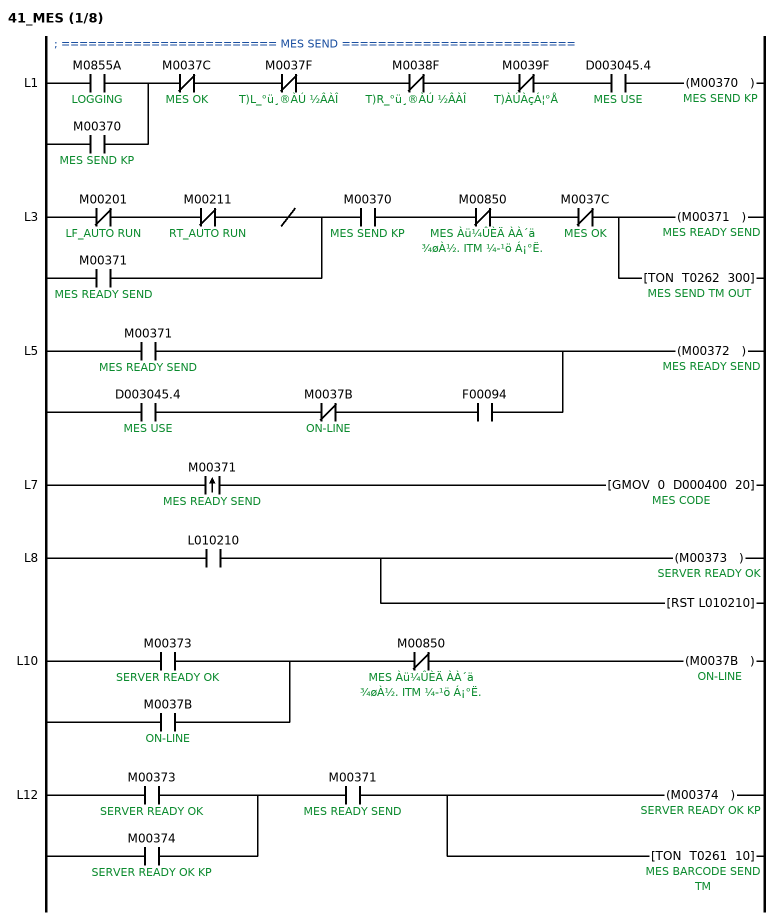
[picture p240: 41_MES rungs L1-L12]
// ======================== MES SEND ==========================
; L1
LOAD      M0855A	// LOGGING
OR        M00370	// MES SEND KP
AND NOT   M0037C	// MES OK
AND NOT   M0037F	// T)L_°ü¸®ÀÚ ½ÂÀÎ
AND NOT   M0038F	// T)R_°ü¸®ÀÚ ½ÂÀÎ
AND NOT   M0039F	// T)ÀÚÀçÁ¦°Å
AND       D003045.4	// MES USE
OUT       M00370	// MES SEND KP
; L3
LOAD NOT  M00201	// LF_AUTO RUN
AND NOT   M00211	// RT_AUTO RUN
NOT
OR        M00371	// MES READY SEND
AND       M00370	// MES SEND KP
AND NOT   M00850	// MES Àü¼ÛÈÄ ÀÀ´ä ¾øÀ½. ITM ¼­¹ö Á¡°Ë.
AND NOT   M0037C	// MES OK
OUT       M00371	// MES READY SEND
TON       T0262 300	// MES SEND TM OUT
; L5
LOAD      M00371	// MES READY SEND
LOAD      D003045.4	// MES USE
AND NOT   M0037B	// ON-LINE
AND       F00094
OR LOAD
OUT       M00372	// MES READY SEND
; L7
LOADP     M00371	// MES READY SEND
GMOV      0 D000400 20	// MES CODE
; L8
LOAD      L010210
OUT       M00373	// SERVER READY OK
RST       L010210
; L10
LOAD      M00373	// SERVER READY OK
OR        M0037B	// ON-LINE
AND NOT   M00850	// MES Àü¼ÛÈÄ ÀÀ´ä ¾øÀ½. ITM ¼­¹ö Á¡°Ë.
OUT       M0037B	// ON-LINE
; L12
LOAD      M00373	// SERVER READY OK
OR        M00374	// SERVER READY OK KP
AND       M00371	// MES READY SEND
OUT       M00374	// SERVER READY OK KP
TON       T0261 10	// MES BARCODE SEND TM

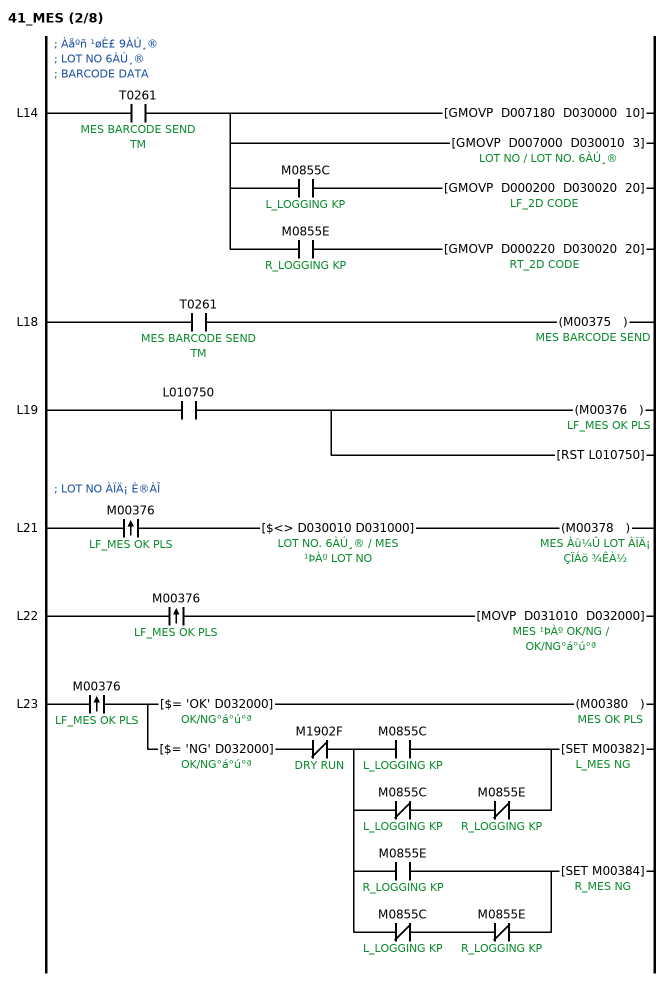
; L14
LOAD      T0261	// MES BARCODE SEND TM
GMOVP     D007180 D030000 10
GMOVP     D007000 D030010 3	// LOT NO / LOT NO. 6ÀÚ¸®
MPUSH
AND       M0855C	// L_LOGGING KP
GMOVP     D000200 D030020 20	// LF_2D CODE
MPOP
AND       M0855E	// R_LOGGING KP
GMOVP     D000220 D030020 20	// RT_2D CODE
// output comment: Àåºñ ¹øÈ£ 9ÀÚ¸®
// output comment: LOT NO 6ÀÚ¸®
// output comment: BARCODE DATA
; L18
LOAD      T0261	// MES BARCODE SEND TM
OUT       M00375	// MES BARCODE SEND
; L19
LOAD      L010750
OUT       M00376	// LF_MES OK PLS
RST       L010750
; L21
LOADP     M00376	// LF_MES OK PLS
AND$<>    D030010 D031000	// LOT NO. 6ÀÚ¸® / MES ¹ÞÀº LOT NO
OUT       M00378	// MES Àü¼Û LOT ÀÏÄ¡ ÇÏÁö ¾ÊÀ½
// output comment: LOT NO ÀÏÄ¡ È®ÀÎ
; L22
LOADP     M00376	// LF_MES OK PLS
MOVP      D031010 D032000	// MES ¹ÞÀº OK/NG / OK/NG°á°ú°ª
; L23
LOADP     M00376	// LF_MES OK PLS
MPUSH
AND$=     'OK' D032000	// OK/NG°á°ú°ª
OUT       M00380	// MES OK PLS
MPOP
AND$=     'NG' D032000	// OK/NG°á°ú°ª
AND NOT   M1902F	// DRY RUN
MPUSH
LOAD      M0855C	// L_LOGGING KP
LOAD NOT  M0855C	// L_LOGGING KP
AND NOT   M0855E	// R_LOGGING KP
OR LOAD
AND LOAD
SET       M00382	// L_MES NG
MPOP
LOAD      M0855E	// R_LOGGING KP
LOAD NOT  M0855C	// L_LOGGING KP
AND NOT   M0855E	// R_LOGGING KP
OR LOAD
AND LOAD
SET       M00384	// R_MES NG

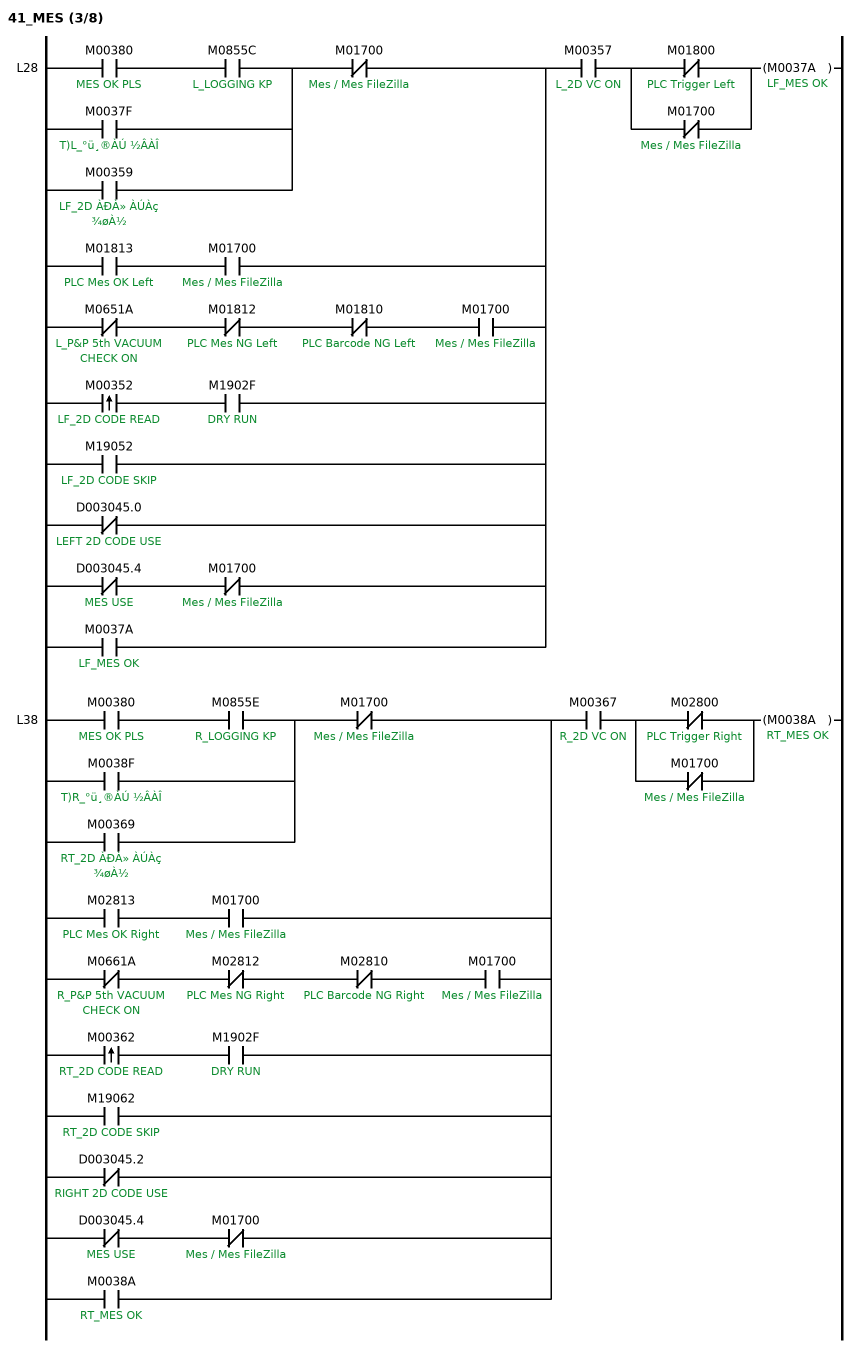
; L28
LOAD      M00380	// MES OK PLS
AND       M0855C	// L_LOGGING KP
OR        M0037F	// T)L_°ü¸®ÀÚ ½ÂÀÎ
OR        M00359	// LF_2D ÀÐÀ» ÀÚÀç ¾øÀ½
AND NOT   M01700	// Mes / Mes FileZilla
LOAD      M01813	// PLC Mes OK Left
AND       M01700	// Mes / Mes FileZilla
OR LOAD
LOAD NOT  M0651A	// L_P&P 5th VACUUM CHECK ON
AND NOT   M01812	// PLC Mes NG Left
AND NOT   M01810	// PLC Barcode NG Left
AND       M01700	// Mes / Mes FileZilla
OR LOAD
LOADP     M00352	// LF_2D CODE READ
AND       M1902F	// DRY RUN
OR LOAD
OR        M19052	// LF_2D CODE SKIP
OR NOT    D003045.0	// LEFT 2D CODE USE
LOAD NOT  D003045.4	// MES USE
AND NOT   M01700	// Mes / Mes FileZilla
OR LOAD
OR        M0037A	// LF_MES OK
AND       M00357	// L_2D VC ON
LOAD NOT  M01800	// PLC Trigger Left
OR NOT    M01700	// Mes / Mes FileZilla
AND LOAD
OUT       M0037A	// LF_MES OK
; L38
LOAD      M00380	// MES OK PLS
AND       M0855E	// R_LOGGING KP
OR        M0038F	// T)R_°ü¸®ÀÚ ½ÂÀÎ
OR        M00369	// RT_2D ÀÐÀ» ÀÚÀç ¾øÀ½
AND NOT   M01700	// Mes / Mes FileZilla
LOAD      M02813	// PLC Mes OK Right
AND       M01700	// Mes / Mes FileZilla
OR LOAD
LOAD NOT  M0661A	// R_P&P 5th VACUUM CHECK ON
AND NOT   M02812	// PLC Mes NG Right
AND NOT   M02810	// PLC Barcode NG Right
AND       M01700	// Mes / Mes FileZilla
OR LOAD
LOADP     M00362	// RT_2D CODE READ
AND       M1902F	// DRY RUN
OR LOAD
OR        M19062	// RT_2D CODE SKIP
OR NOT    D003045.2	// RIGHT 2D CODE USE
LOAD NOT  D003045.4	// MES USE
AND NOT   M01700	// Mes / Mes FileZilla
OR LOAD
OR        M0038A	// RT_MES OK
AND       M00367	// R_2D VC ON
LOAD NOT  M02800	// PLC Trigger Right
OR NOT    M01700	// Mes / Mes FileZilla
AND LOAD
OUT       M0038A	// RT_MES OK

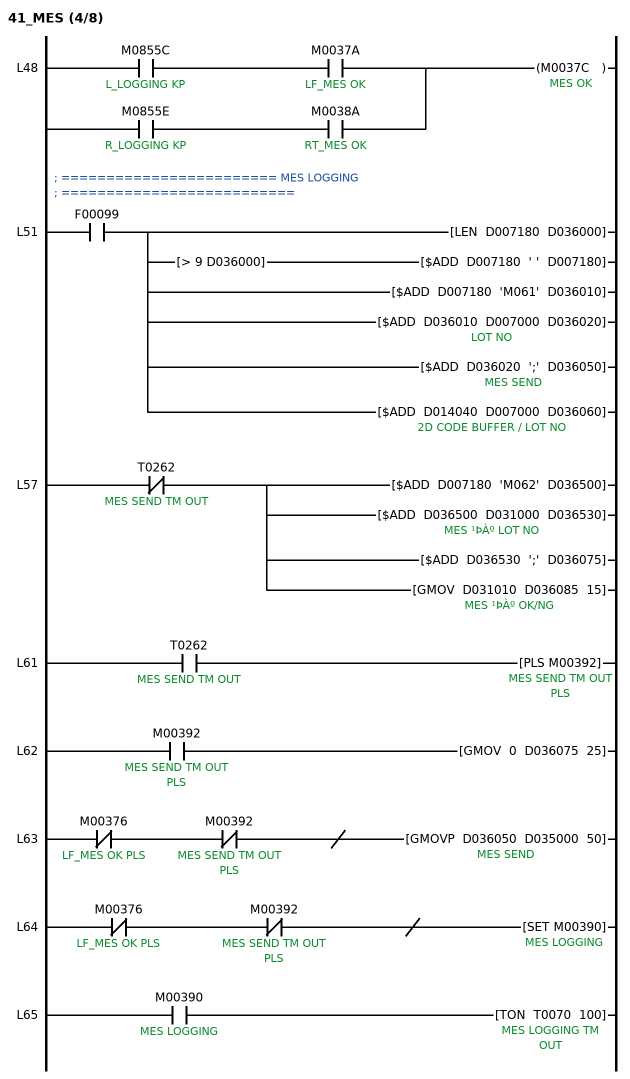
; L48
LOAD      M0855C	// L_LOGGING KP
AND       M0037A	// LF_MES OK
LOAD      M0855E	// R_LOGGING KP
AND       M0038A	// RT_MES OK
OR LOAD
OUT       M0037C	// MES OK
// ======================== MES LOGGING ==========================
; L51
LOAD      F00099
LEN       D007180 D036000
MPUSH
AND>      9 D036000
$ADD      D007180 ' ' D007180
MPOP
$ADD      D007180 'M061' D036010
$ADD      D036010 D007000 D036020	// LOT NO
$ADD      D036020 ';' D036050	// MES SEND
$ADD      D014040 D007000 D036060	// 2D CODE BUFFER / LOT NO
; L57
LOAD NOT  T0262	// MES SEND TM OUT
$ADD      D007180 'M062' D036500
$ADD      D036500 D031000 D036530	// MES ¹ÞÀº LOT NO
$ADD      D036530 ';' D036075
GMOV      D031010 D036085 15	// MES ¹ÞÀº OK/NG
; L61
LOAD      T0262	// MES SEND TM OUT
OUTP      M00392	// MES SEND TM OUT PLS
; L62
LOAD      M00392	// MES SEND TM OUT PLS
GMOV      0 D036075 25
; L63
LOAD NOT  M00376	// LF_MES OK PLS
AND NOT   M00392	// MES SEND TM OUT PLS
NOT
GMOVP     D036050 D035000 50	// MES SEND
; L64
LOAD NOT  M00376	// LF_MES OK PLS
AND NOT   M00392	// MES SEND TM OUT PLS
NOT
SET       M00390	// MES LOGGING
; L65
LOAD      M00390	// MES LOGGING
TON       T0070 100	// MES LOGGING TM OUT

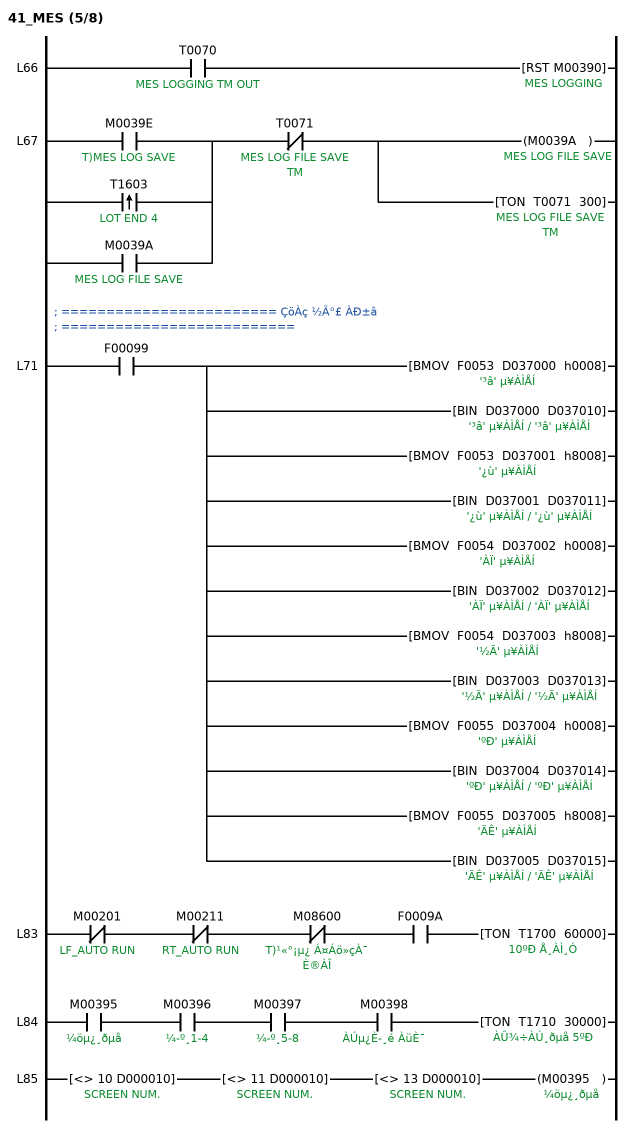
; L66
LOAD      T0070	// MES LOGGING TM OUT
RST       M00390	// MES LOGGING
; L67
LOAD      M0039E	// T)MES LOG SAVE
ORP       T1603	// LOT END 4
OR        M0039A	// MES LOG FILE SAVE
AND NOT   T0071	// MES LOG FILE SAVE TM
OUT       M0039A	// MES LOG FILE SAVE
TON       T0071 300	// MES LOG FILE SAVE TM
// ======================== ÇöÀç ½Ã°£ ÀÐ±â ==========================
; L71
LOAD      F00099
BMOV      F0053 D037000 h0008	// '³â' µ¥ÀÌÅÍ
BIN       D037000 D037010	// '³â' µ¥ÀÌÅÍ / '³â' µ¥ÀÌÅÍ
BMOV      F0053 D037001 h8008	// '¿ù' µ¥ÀÌÅÍ
BIN       D037001 D037011	// '¿ù' µ¥ÀÌÅÍ / '¿ù' µ¥ÀÌÅÍ
BMOV      F0054 D037002 h0008	// 'ÀÏ' µ¥ÀÌÅÍ
BIN       D037002 D037012	// 'ÀÏ' µ¥ÀÌÅÍ / 'ÀÏ' µ¥ÀÌÅÍ
BMOV      F0054 D037003 h8008	// '½Ã' µ¥ÀÌÅÍ
BIN       D037003 D037013	// '½Ã' µ¥ÀÌÅÍ / '½Ã' µ¥ÀÌÅÍ
BMOV      F0055 D037004 h0008	// 'ºÐ' µ¥ÀÌÅÍ
BIN       D037004 D037014	// 'ºÐ' µ¥ÀÌÅÍ / 'ºÐ' µ¥ÀÌÅÍ
BMOV      F0055 D037005 h8008	// 'ÃÊ' µ¥ÀÌÅÍ
BIN       D037005 D037015	// 'ÃÊ' µ¥ÀÌÅÍ / 'ÃÊ' µ¥ÀÌÅÍ
; L83
LOAD NOT  M00201	// LF_AUTO RUN
AND NOT   M00211	// RT_AUTO RUN
AND NOT   M08600	// T)¹«°¡µ¿ Á¤Áö»çÀ¯ È®ÀÎ
AND       F0009A
TON       T1700 60000	// 10ºÐ Å¸ÀÌ¸Ó
; L84
LOAD      M00395	// ¼öµ¿¸ðµå
AND       M00396	// ¼­º¸1-4
AND       M00397	// ¼­º¸5-8
AND       M00398	// ÀÚµ¿È­¸é ÀüÈ¯
TON       T1710 30000	// ÀÛ¾÷ÀÚ¸ðµå 5ºÐ
; L85
LOAD<>    10 D000010	// SCREEN NUM.
AND<>     11 D000010	// SCREEN NUM.
AND<>     13 D000010	// SCREEN NUM.
OUT       M00395	// ¼öµ¿¸ðµå

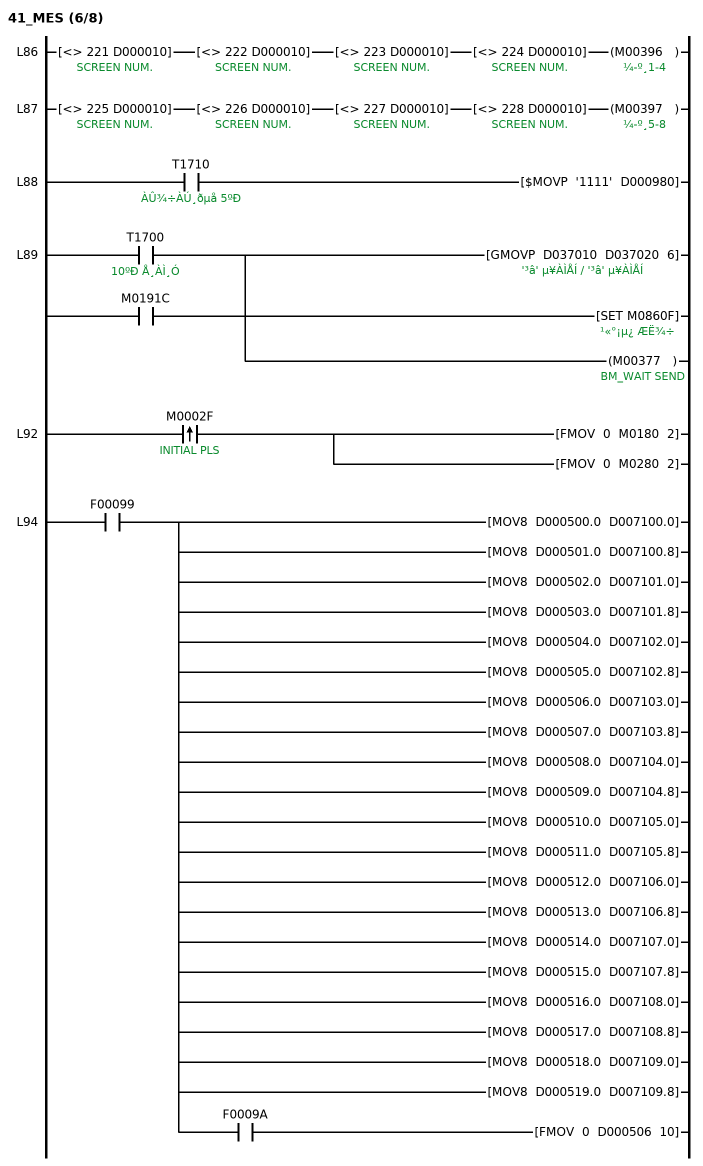
; L86
LOAD<>    221 D000010	// SCREEN NUM.
AND<>     222 D000010	// SCREEN NUM.
AND<>     223 D000010	// SCREEN NUM.
AND<>     224 D000010	// SCREEN NUM.
OUT       M00396	// ¼­º¸1-4
; L87
LOAD<>    225 D000010	// SCREEN NUM.
AND<>     226 D000010	// SCREEN NUM.
AND<>     227 D000010	// SCREEN NUM.
AND<>     228 D000010	// SCREEN NUM.
OUT       M00397	// ¼­º¸5-8
; L88
LOAD      T1710	// ÀÛ¾÷ÀÚ¸ðµå 5ºÐ
$MOVP     '1111' D000980
; L89
LOAD      T1700	// 10ºÐ Å¸ÀÌ¸Ó
OR        M0191C
GMOVP     D037010 D037020 6	// '³â' µ¥ÀÌÅÍ / '³â' µ¥ÀÌÅÍ
SET       M0860F	// ¹«°¡µ¿ ÆË¾÷
OUT       M00377	// BM_WAIT SEND
; L92
LOADP     M0002F	// INITIAL PLS
FMOV      0 M0180 2
FMOV      0 M0280 2
; L94
LOAD      F00099
MOV8      D000500.0 D007100.0
MOV8      D000501.0 D007100.8
MOV8      D000502.0 D007101.0
MOV8      D000503.0 D007101.8
MOV8      D000504.0 D007102.0
MOV8      D000505.0 D007102.8
MOV8      D000506.0 D007103.0
MOV8      D000507.0 D007103.8
MOV8      D000508.0 D007104.0
MOV8      D000509.0 D007104.8
MOV8      D000510.0 D007105.0
MOV8      D000511.0 D007105.8
MOV8      D000512.0 D007106.0
MOV8      D000513.0 D007106.8
MOV8      D000514.0 D007107.0
MOV8      D000515.0 D007107.8
MOV8      D000516.0 D007108.0
MOV8      D000517.0 D007108.8
MOV8      D000518.0 D007109.0
MOV8      D000519.0 D007109.8
AND       F0009A
FMOV      0 D000506 10

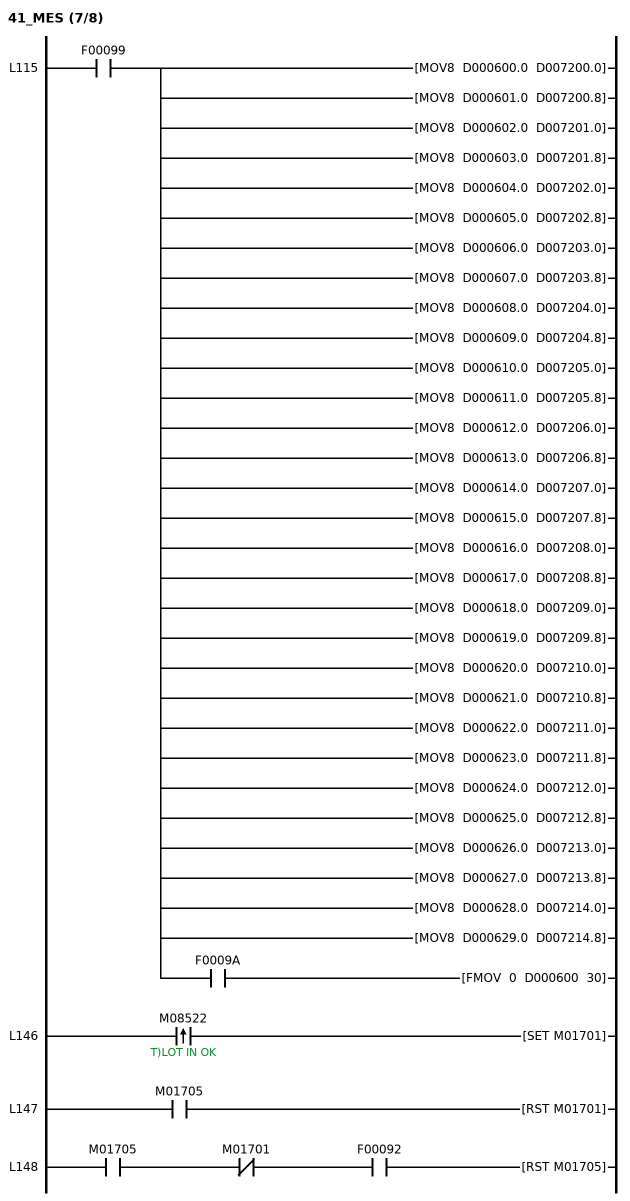
; L115
LOAD      F00099
MOV8      D000600.0 D007200.0
MOV8      D000601.0 D007200.8
MOV8      D000602.0 D007201.0
MOV8      D000603.0 D007201.8
MOV8      D000604.0 D007202.0
MOV8      D000605.0 D007202.8
MOV8      D000606.0 D007203.0
MOV8      D000607.0 D007203.8
MOV8      D000608.0 D007204.0
MOV8      D000609.0 D007204.8
MOV8      D000610.0 D007205.0
MOV8      D000611.0 D007205.8
MOV8      D000612.0 D007206.0
MOV8      D000613.0 D007206.8
MOV8      D000614.0 D007207.0
MOV8      D000615.0 D007207.8
MOV8      D000616.0 D007208.0
MOV8      D000617.0 D007208.8
MOV8      D000618.0 D007209.0
MOV8      D000619.0 D007209.8
MOV8      D000620.0 D007210.0
MOV8      D000621.0 D007210.8
MOV8      D000622.0 D007211.0
MOV8      D000623.0 D007211.8
MOV8      D000624.0 D007212.0
MOV8      D000625.0 D007212.8
MOV8      D000626.0 D007213.0
MOV8      D000627.0 D007213.8
MOV8      D000628.0 D007214.0
MOV8      D000629.0 D007214.8
AND       F0009A
FMOV      0 D000600 30
; L146
LOADP     M08522	// T)LOT IN OK
SET       M01701
; L147
LOAD      M01705
RST       M01701
; L148
LOAD      M01705
AND NOT   M01701
AND       F00092
RST       M01705

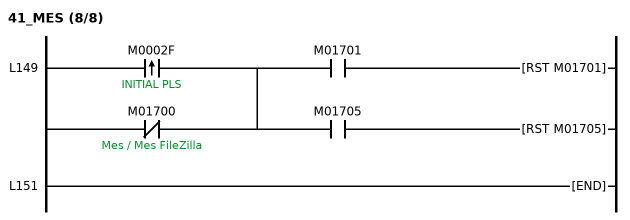
; L149
LOADP     M0002F	// INITIAL PLS
OR NOT    M01700	// Mes / Mes FileZilla
MPUSH
AND       M01701
RST       M01701
MPOP
AND       M01705
RST       M01705
; L151
END

PROGRAM 51_MT_01_2_3_4 (task: ½ºÄµ ÇÁ·Î±×·¥)

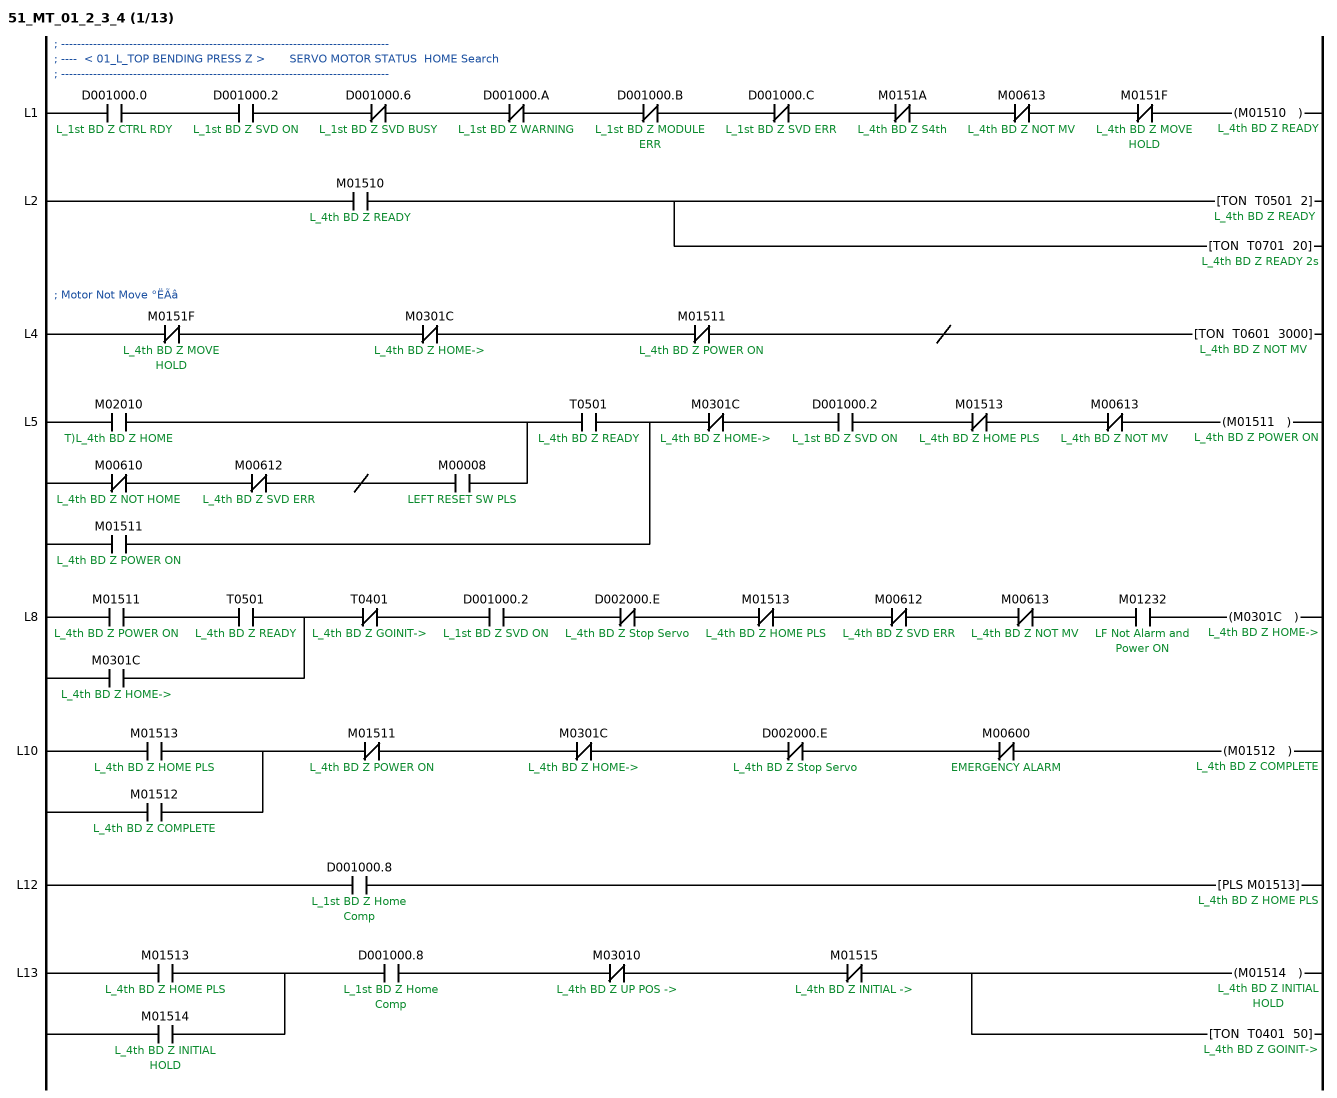
// ----------------------------------------------------------------------------------
// 
// ----  < 01_L_TOP BENDING PRESS Z >       SERVO MOTOR STATUS  HOME Search
// 
// ----------------------------------------------------------------------------------
; L1
LOAD      D001000.0	// L_1st BD Z CTRL RDY
AND       D001000.2	// L_1st BD Z SVD ON
AND NOT   D001000.6	// L_1st BD Z SVD BUSY
AND NOT   D001000.A	// L_1st BD Z WARNING
AND NOT   D001000.B	// L_1st BD Z MODULE ERR
AND NOT   D001000.C	// L_1st BD Z SVD ERR
AND NOT   M0151A	// L_4th BD Z S4th
AND NOT   M00613	// L_4th BD Z NOT MV
AND NOT   M0151F	// L_4th BD Z MOVE HOLD
OUT       M01510	// L_4th BD Z READY
; L2
LOAD      M01510	// L_4th BD Z READY
TON       T0501 2	// L_4th BD Z READY
TON       T0701 20	// L_4th BD Z READY 2s
; L4
LOAD NOT  M0151F	// L_4th BD Z MOVE HOLD
AND NOT   M0301C	// L_4th BD Z HOME->
AND NOT   M01511	// L_4th BD Z POWER ON
NOT
TON       T0601 3000	// L_4th BD Z NOT MV
// output comment: Motor Not Move °ËÃâ
; L5
LOAD      M02010	// T)L_4th BD Z HOME
LOAD NOT  M00610	// L_4th BD Z NOT HOME
AND NOT   M00612	// L_4th BD Z SVD ERR
NOT
AND       M00008	// LEFT RESET SW PLS
OR LOAD
AND       T0501	// L_4th BD Z READY
OR        M01511	// L_4th BD Z POWER ON
AND NOT   M0301C	// L_4th BD Z HOME->
AND       D001000.2	// L_1st BD Z SVD ON
AND NOT   M01513	// L_4th BD Z HOME PLS
AND NOT   M00613	// L_4th BD Z NOT MV
OUT       M01511	// L_4th BD Z POWER ON
; L8
LOAD      M01511	// L_4th BD Z POWER ON
AND       T0501	// L_4th BD Z READY
OR        M0301C	// L_4th BD Z HOME->
AND NOT   T0401	// L_4th BD Z GOINIT->
AND       D001000.2	// L_1st BD Z SVD ON
AND NOT   D002000.E	// L_4th BD Z Stop Servo
AND NOT   M01513	// L_4th BD Z HOME PLS
AND NOT   M00612	// L_4th BD Z SVD ERR
AND NOT   M00613	// L_4th BD Z NOT MV
AND       M01232	// LF Not Alarm and Power ON
OUT       M0301C	// L_4th BD Z HOME->
; L10
LOAD      M01513	// L_4th BD Z HOME PLS
OR        M01512	// L_4th BD Z COMPLETE
AND NOT   M01511	// L_4th BD Z POWER ON
AND NOT   M0301C	// L_4th BD Z HOME->
AND NOT   D002000.E	// L_4th BD Z Stop Servo
AND NOT   M00600	// EMERGENCY ALARM
OUT       M01512	// L_4th BD Z COMPLETE
; L12
LOAD      D001000.8	// L_1st BD Z Home Comp
OUTP      M01513	// L_4th BD Z HOME PLS
; L13
LOAD      M01513	// L_4th BD Z HOME PLS
OR        M01514	// L_4th BD Z INITIAL HOLD
AND       D001000.8	// L_1st BD Z Home Comp
AND NOT   M03010	// L_4th BD Z UP POS ->
AND NOT   M01515	// L_4th BD Z INITIAL ->
OUT       M01514	// L_4th BD Z INITIAL HOLD
TON       T0401 50	// L_4th BD Z GOINIT->

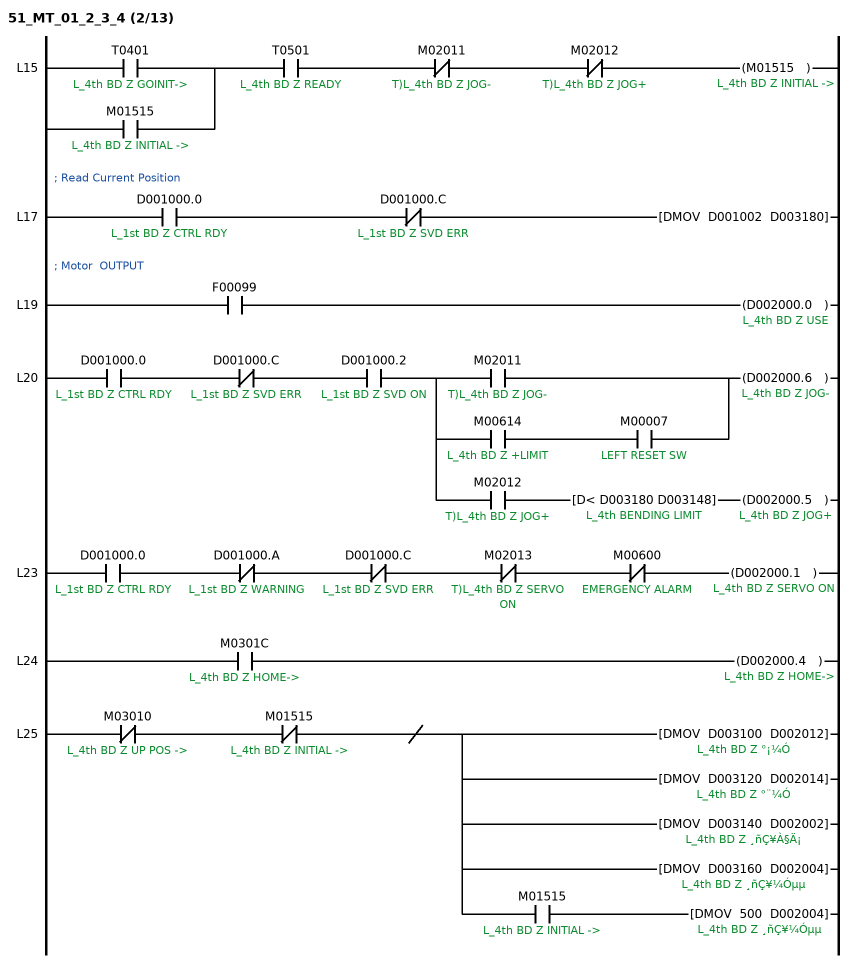
; L15
LOAD      T0401	// L_4th BD Z GOINIT->
OR        M01515	// L_4th BD Z INITIAL ->
AND       T0501	// L_4th BD Z READY
AND NOT   M02011	// T)L_4th BD Z JOG-
AND NOT   M02012	// T)L_4th BD Z JOG+
OUT       M01515	// L_4th BD Z INITIAL ->
; L17
LOAD      D001000.0	// L_1st BD Z CTRL RDY
AND NOT   D001000.C	// L_1st BD Z SVD ERR
DMOV      D001002 D003180
// output comment: Read Current Position
//  Motor  OUTPUT
; L19
LOAD      F00099
OUT       D002000.0	// L_4th BD Z USE
; L20
LOAD      D001000.0	// L_1st BD Z CTRL RDY
AND NOT   D001000.C	// L_1st BD Z SVD ERR
AND       D001000.2	// L_1st BD Z SVD ON
MPUSH
LOAD      M02011	// T)L_4th BD Z JOG-
LOAD      M00614	// L_4th BD Z +LIMIT
AND       M00007	// LEFT RESET SW
OR LOAD
AND LOAD
OUT       D002000.6	// L_4th BD Z JOG-
MPOP
AND       M02012	// T)L_4th BD Z JOG+
ANDD<     D003180 D003148	// L_4th BENDING LIMIT
OUT       D002000.5	// L_4th BD Z JOG+
; L23
LOAD      D001000.0	// L_1st BD Z CTRL RDY
AND NOT   D001000.A	// L_1st BD Z WARNING
AND NOT   D001000.C	// L_1st BD Z SVD ERR
AND NOT   M02013	// T)L_4th BD Z SERVO ON
AND NOT   M00600	// EMERGENCY ALARM
OUT       D002000.1	// L_4th BD Z SERVO ON
; L24
LOAD      M0301C	// L_4th BD Z HOME->
OUT       D002000.4	// L_4th BD Z HOME->
; L25
LOAD NOT  M03010	// L_4th BD Z UP POS ->
AND NOT   M01515	// L_4th BD Z INITIAL ->
NOT
DMOV      D003100 D002012	// L_4th BD Z °¡¼Ó
DMOV      D003120 D002014	// L_4th BD Z °¨¼Ó
DMOV      D003140 D002002	// L_4th BD Z ¸ñÇ¥À§Ä¡
DMOV      D003160 D002004	// L_4th BD Z ¸ñÇ¥¼Óµµ
AND       M01515	// L_4th BD Z INITIAL ->
DMOV      500 D002004	// L_4th BD Z ¸ñÇ¥¼Óµµ

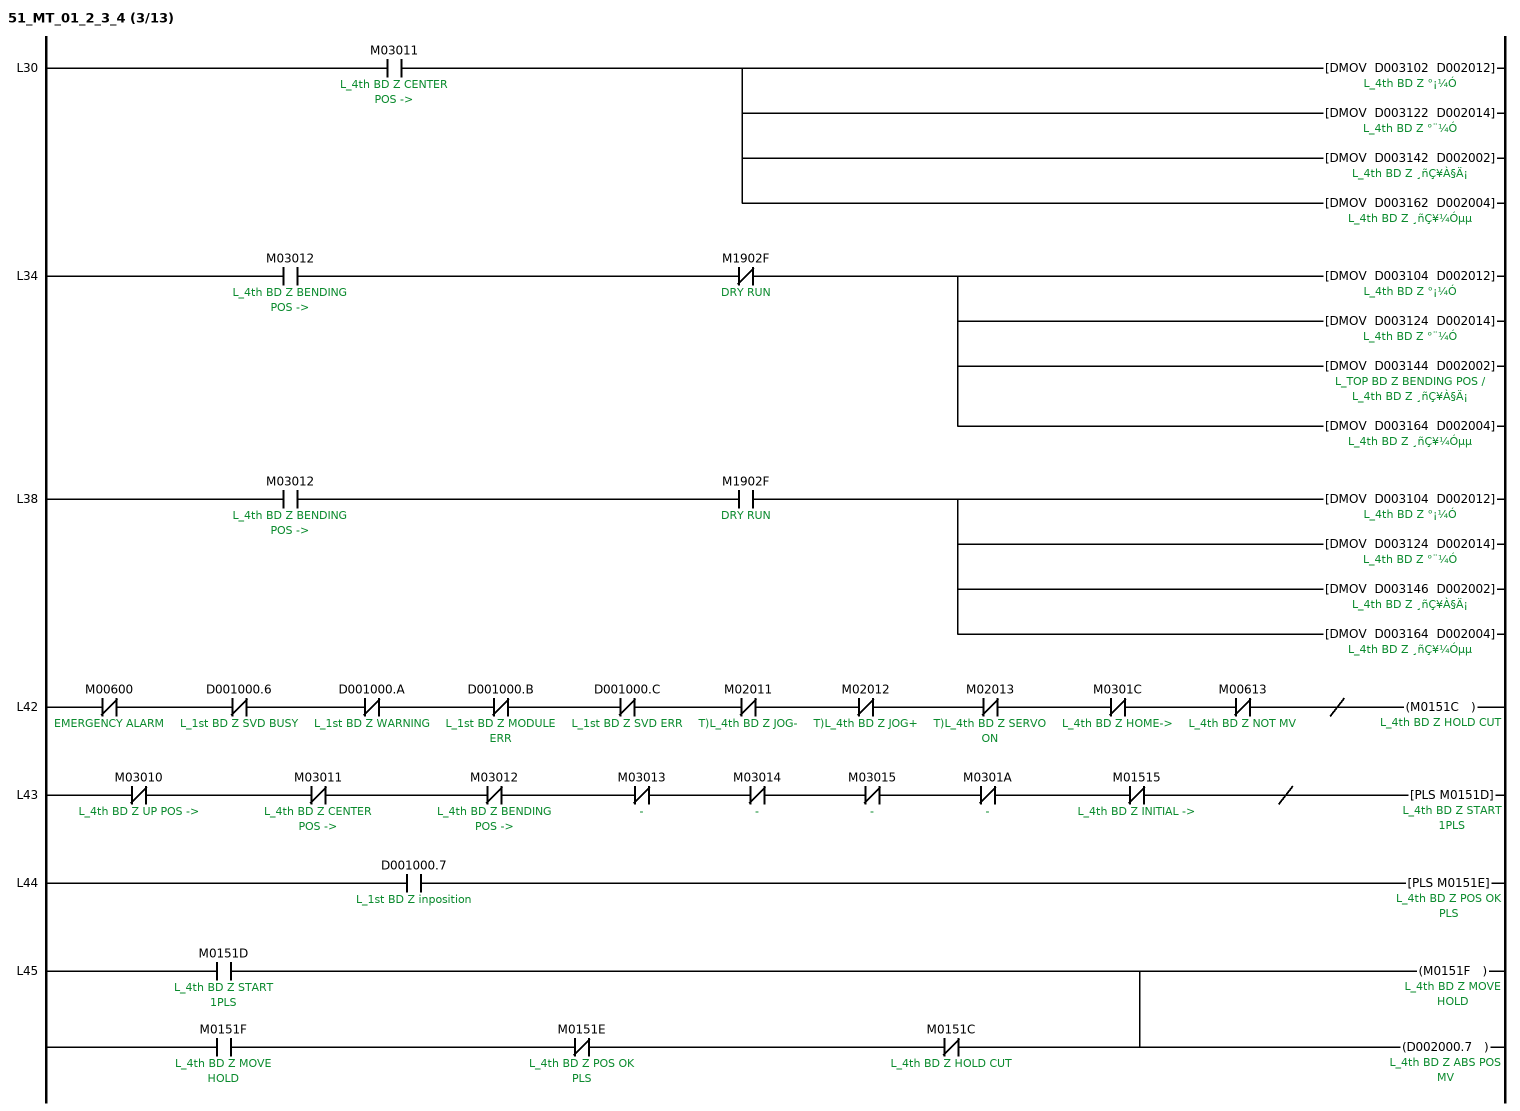
; L30
LOAD      M03011	// L_4th BD Z CENTER POS ->
DMOV      D003102 D002012	// L_4th BD Z °¡¼Ó
DMOV      D003122 D002014	// L_4th BD Z °¨¼Ó
DMOV      D003142 D002002	// L_4th BD Z ¸ñÇ¥À§Ä¡
DMOV      D003162 D002004	// L_4th BD Z ¸ñÇ¥¼Óµµ
; L34
LOAD      M03012	// L_4th BD Z BENDING POS ->
AND NOT   M1902F	// DRY RUN
DMOV      D003104 D002012	// L_4th BD Z °¡¼Ó
DMOV      D003124 D002014	// L_4th BD Z °¨¼Ó
DMOV      D003144 D002002	// L_TOP BD Z BENDING POS / L_4th BD Z ¸ñÇ¥À§Ä¡
DMOV      D003164 D002004	// L_4th BD Z ¸ñÇ¥¼Óµµ
; L38
LOAD      M03012	// L_4th BD Z BENDING POS ->
AND       M1902F	// DRY RUN
DMOV      D003104 D002012	// L_4th BD Z °¡¼Ó
DMOV      D003124 D002014	// L_4th BD Z °¨¼Ó
DMOV      D003146 D002002	// L_4th BD Z ¸ñÇ¥À§Ä¡
DMOV      D003164 D002004	// L_4th BD Z ¸ñÇ¥¼Óµµ
; L42
LOAD NOT  M00600	// EMERGENCY ALARM
AND NOT   D001000.6	// L_1st BD Z SVD BUSY
AND NOT   D001000.A	// L_1st BD Z WARNING
AND NOT   D001000.B	// L_1st BD Z MODULE ERR
AND NOT   D001000.C	// L_1st BD Z SVD ERR
AND NOT   M02011	// T)L_4th BD Z JOG-
AND NOT   M02012	// T)L_4th BD Z JOG+
AND NOT   M02013	// T)L_4th BD Z SERVO ON
AND NOT   M0301C	// L_4th BD Z HOME->
AND NOT   M00613	// L_4th BD Z NOT MV
NOT
OUT       M0151C	// L_4th BD Z HOLD CUT
; L43
LOAD NOT  M03010	// L_4th BD Z UP POS ->
AND NOT   M03011	// L_4th BD Z CENTER POS ->
AND NOT   M03012	// L_4th BD Z BENDING POS ->
AND NOT   M03013	// -
AND NOT   M03014	// -
AND NOT   M03015	// -
AND NOT   M0301A	// -
AND NOT   M01515	// L_4th BD Z INITIAL ->
NOT
OUTP      M0151D	// L_4th BD Z START 1PLS
; L44
LOAD      D001000.7	// L_1st BD Z inposition
OUTP      M0151E	// L_4th BD Z POS OK PLS
; L45
LOAD      M0151D	// L_4th BD Z START 1PLS
LOAD      M0151F	// L_4th BD Z MOVE HOLD
AND NOT   M0151E	// L_4th BD Z POS OK PLS
AND NOT   M0151C	// L_4th BD Z HOLD CUT
OR LOAD
OUT       M0151F	// L_4th BD Z MOVE HOLD
OUT       D002000.7	// L_4th BD Z ABS POS MV

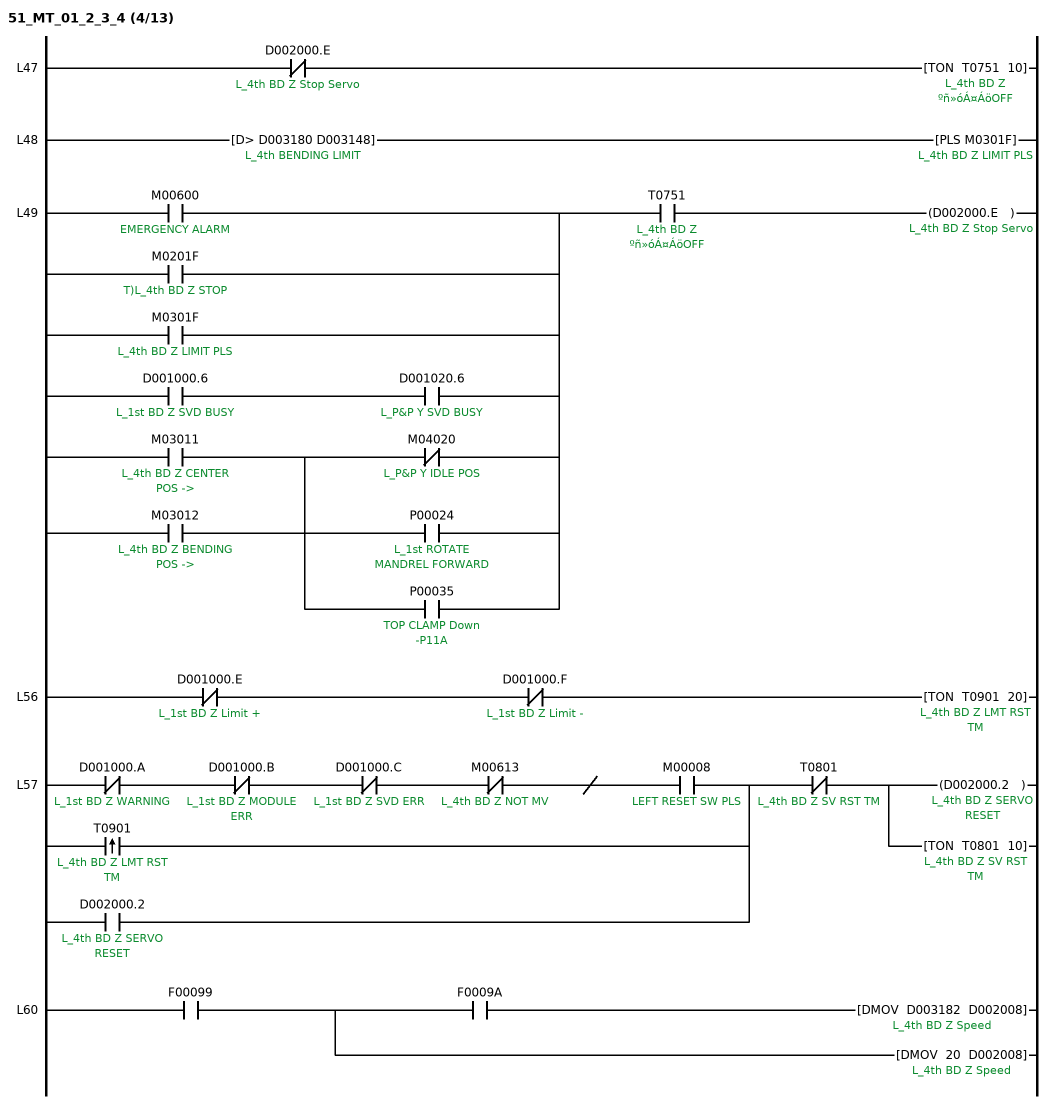
; L47
LOAD NOT  D002000.E	// L_4th BD Z Stop Servo
TON       T0751 10	// L_4th BD Z ºñ»óÁ¤ÁöOFF
; L48
LOADD>    D003180 D003148	// L_4th BENDING LIMIT
OUTP      M0301F	// L_4th BD Z LIMIT PLS
; L49
LOAD      M00600	// EMERGENCY ALARM
OR        M0201F	// T)L_4th BD Z STOP
OR        M0301F	// L_4th BD Z LIMIT PLS
LOAD      D001000.6	// L_1st BD Z SVD BUSY
AND       D001020.6	// L_P&P Y SVD BUSY
OR LOAD
LOAD      M03011	// L_4th BD Z CENTER POS ->
OR        M03012	// L_4th BD Z BENDING POS ->
LOAD NOT  M04020	// L_P&P Y IDLE POS
OR        P00024	// L_1st ROTATE MANDREL FORWARD
OR        P00035	// TOP CLAMP Down -P11A
AND LOAD
OR LOAD
AND       T0751	// L_4th BD Z ºñ»óÁ¤ÁöOFF
OUT       D002000.E	// L_4th BD Z Stop Servo
; L56
LOAD NOT  D001000.E	// L_1st BD Z Limit +
AND NOT   D001000.F	// L_1st BD Z Limit -
TON       T0901 20	// L_4th BD Z LMT RST TM
; L57
LOAD NOT  D001000.A	// L_1st BD Z WARNING
AND NOT   D001000.B	// L_1st BD Z MODULE ERR
AND NOT   D001000.C	// L_1st BD Z SVD ERR
AND NOT   M00613	// L_4th BD Z NOT MV
NOT
AND       M00008	// LEFT RESET SW PLS
ORP       T0901	// L_4th BD Z LMT RST TM
OR        D002000.2	// L_4th BD Z SERVO RESET
AND NOT   T0801	// L_4th BD Z SV RST TM
OUT       D002000.2	// L_4th BD Z SERVO RESET
TON       T0801 10	// L_4th BD Z SV RST TM
; L60
LOAD      F00099
MPUSH
AND       F0009A
DMOV      D003182 D002008	// L_4th BD Z Speed
MPOP
DMOV      20 D002008	// L_4th BD Z Speed

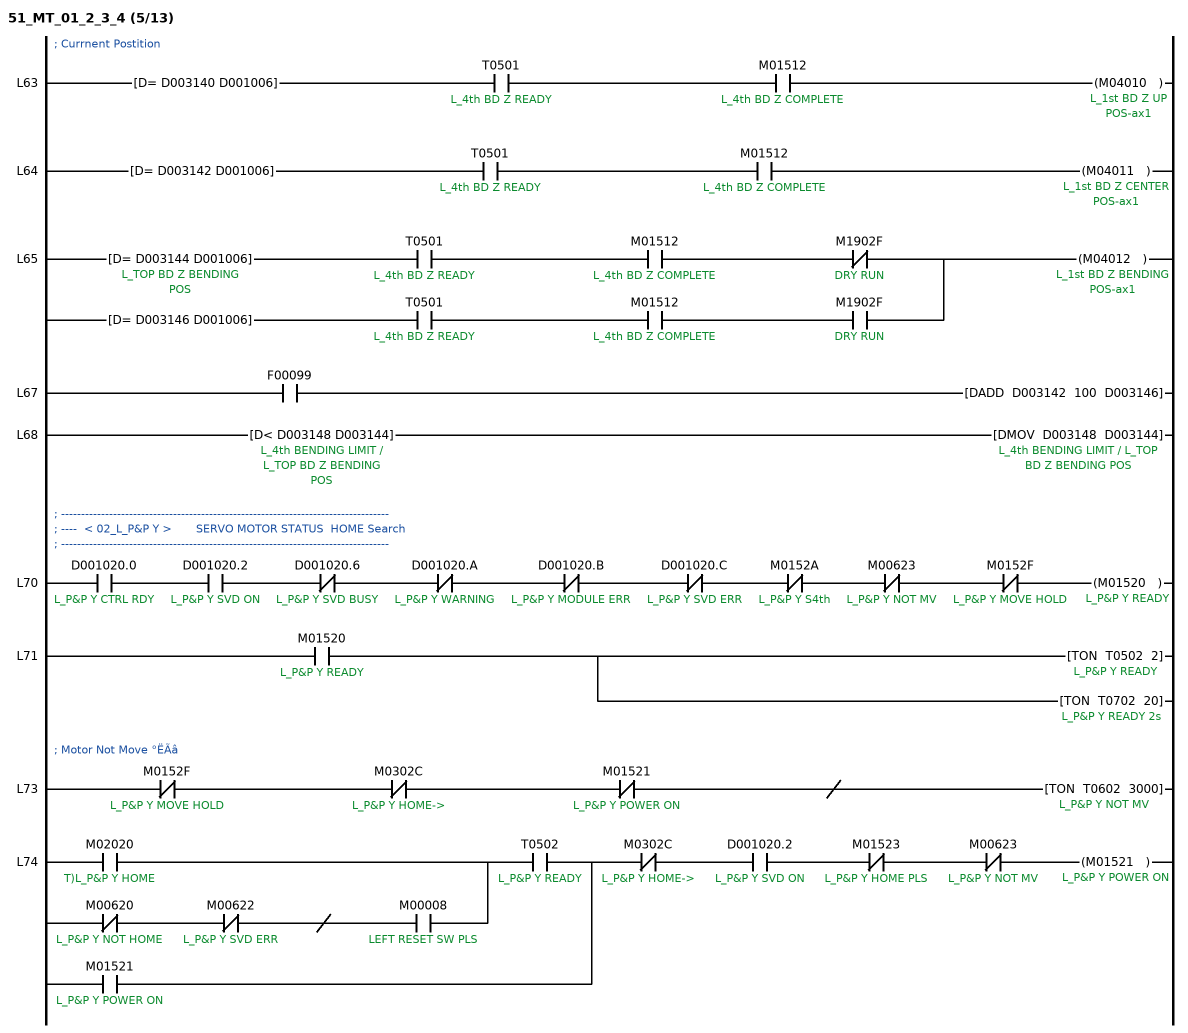
// Currnent Postition
; L63
LOADD=    D003140 D001006
AND       T0501	// L_4th BD Z READY
AND       M01512	// L_4th BD Z COMPLETE
OUT       M04010	// L_1st BD Z UP POS-ax1
; L64
LOADD=    D003142 D001006
AND       T0501	// L_4th BD Z READY
AND       M01512	// L_4th BD Z COMPLETE
OUT       M04011	// L_1st BD Z CENTER POS-ax1
; L65
LOADD=    D003144 D001006	// L_TOP BD Z BENDING POS
AND       T0501	// L_4th BD Z READY
AND       M01512	// L_4th BD Z COMPLETE
AND NOT   M1902F	// DRY RUN
LOADD=    D003146 D001006
AND       T0501	// L_4th BD Z READY
AND       M01512	// L_4th BD Z COMPLETE
AND       M1902F	// DRY RUN
OR LOAD
OUT       M04012	// L_1st BD Z BENDING POS-ax1
; L67
LOAD      F00099
DADD      D003142 100 D003146
; L68
LOADD<    D003148 D003144	// L_4th BENDING LIMIT / L_TOP BD Z BENDING POS
DMOV      D003148 D003144	// L_4th BENDING LIMIT / L_TOP BD Z BENDING POS
// ----------------------------------------------------------------------------------
// 
// ----  < 02_L_P&P Y >       SERVO MOTOR STATUS  HOME Search
// 
// ----------------------------------------------------------------------------------
; L70
LOAD      D001020.0	// L_P&P Y CTRL RDY
AND       D001020.2	// L_P&P Y SVD ON
AND NOT   D001020.6	// L_P&P Y SVD BUSY
AND NOT   D001020.A	// L_P&P Y WARNING
AND NOT   D001020.B	// L_P&P Y MODULE ERR
AND NOT   D001020.C	// L_P&P Y SVD ERR
AND NOT   M0152A	// L_P&P Y S4th
AND NOT   M00623	// L_P&P Y NOT MV
AND NOT   M0152F	// L_P&P Y MOVE HOLD
OUT       M01520	// L_P&P Y READY
; L71
LOAD      M01520	// L_P&P Y READY
TON       T0502 2	// L_P&P Y READY
TON       T0702 20	// L_P&P Y READY 2s
; L73
LOAD NOT  M0152F	// L_P&P Y MOVE HOLD
AND NOT   M0302C	// L_P&P Y HOME->
AND NOT   M01521	// L_P&P Y POWER ON
NOT
TON       T0602 3000	// L_P&P Y NOT MV
// output comment: Motor Not Move °ËÃâ
; L74
LOAD      M02020	// T)L_P&P Y HOME
LOAD NOT  M00620	// L_P&P Y NOT HOME
AND NOT   M00622	// L_P&P Y SVD ERR
NOT
AND       M00008	// LEFT RESET SW PLS
OR LOAD
AND       T0502	// L_P&P Y READY
OR        M01521	// L_P&P Y POWER ON
AND NOT   M0302C	// L_P&P Y HOME->
AND       D001020.2	// L_P&P Y SVD ON
AND NOT   M01523	// L_P&P Y HOME PLS
AND NOT   M00623	// L_P&P Y NOT MV
OUT       M01521	// L_P&P Y POWER ON

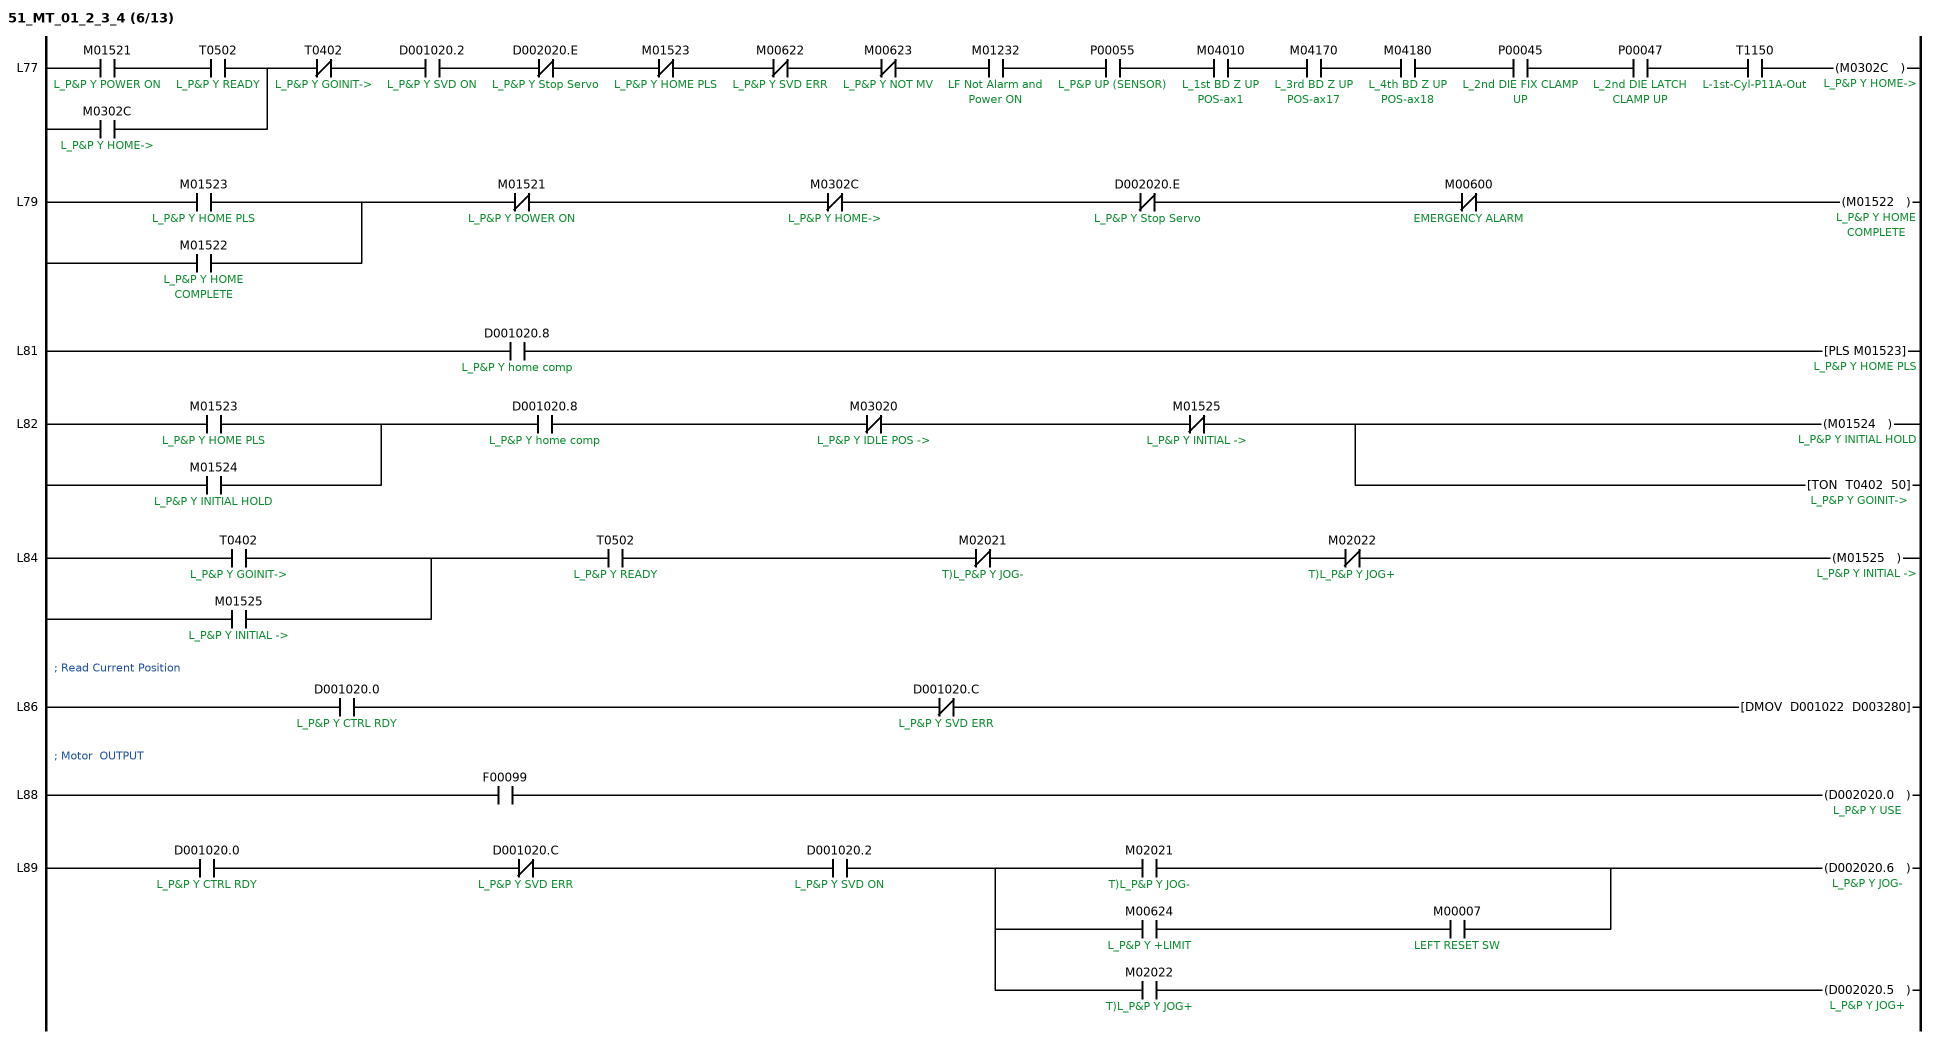
; L77
LOAD      M01521	// L_P&P Y POWER ON
AND       T0502	// L_P&P Y READY
OR        M0302C	// L_P&P Y HOME->
AND NOT   T0402	// L_P&P Y GOINIT->
AND       D001020.2	// L_P&P Y SVD ON
AND NOT   D002020.E	// L_P&P Y Stop Servo
AND NOT   M01523	// L_P&P Y HOME PLS
AND NOT   M00622	// L_P&P Y SVD ERR
AND NOT   M00623	// L_P&P Y NOT MV
AND       M01232	// LF Not Alarm and Power ON
AND       P00055	// L_P&P UP (SENSOR)
AND       M04010	// L_1st BD Z UP POS-ax1
AND       M04170	// L_3rd BD Z UP POS-ax17
AND       M04180	// L_4th BD Z UP POS-ax18
AND       P00045	// L_2nd DIE FIX CLAMP UP
AND       P00047	// L_2nd DIE LATCH CLAMP UP
AND       T1150	// L-1st-Cyl-P11A-Out
OUT       M0302C	// L_P&P Y HOME->
; L79
LOAD      M01523	// L_P&P Y HOME PLS
OR        M01522	// L_P&P Y HOME COMPLETE
AND NOT   M01521	// L_P&P Y POWER ON
AND NOT   M0302C	// L_P&P Y HOME->
AND NOT   D002020.E	// L_P&P Y Stop Servo
AND NOT   M00600	// EMERGENCY ALARM
OUT       M01522	// L_P&P Y HOME COMPLETE
; L81
LOAD      D001020.8	// L_P&P Y home comp
OUTP      M01523	// L_P&P Y HOME PLS
; L82
LOAD      M01523	// L_P&P Y HOME PLS
OR        M01524	// L_P&P Y INITIAL HOLD
AND       D001020.8	// L_P&P Y home comp
AND NOT   M03020	// L_P&P Y IDLE POS ->
AND NOT   M01525	// L_P&P Y INITIAL ->
OUT       M01524	// L_P&P Y INITIAL HOLD
TON       T0402 50	// L_P&P Y GOINIT->
; L84
LOAD      T0402	// L_P&P Y GOINIT->
OR        M01525	// L_P&P Y INITIAL ->
AND       T0502	// L_P&P Y READY
AND NOT   M02021	// T)L_P&P Y JOG-
AND NOT   M02022	// T)L_P&P Y JOG+
OUT       M01525	// L_P&P Y INITIAL ->
; L86
LOAD      D001020.0	// L_P&P Y CTRL RDY
AND NOT   D001020.C	// L_P&P Y SVD ERR
DMOV      D001022 D003280
// output comment: Read Current Position
//  Motor  OUTPUT
; L88
LOAD      F00099
OUT       D002020.0	// L_P&P Y USE
; L89
LOAD      D001020.0	// L_P&P Y CTRL RDY
AND NOT   D001020.C	// L_P&P Y SVD ERR
AND       D001020.2	// L_P&P Y SVD ON
MPUSH
LOAD      M02021	// T)L_P&P Y JOG-
LOAD      M00624	// L_P&P Y +LIMIT
AND       M00007	// LEFT RESET SW
OR LOAD
AND LOAD
OUT       D002020.6	// L_P&P Y JOG-
MPOP
AND       M02022	// T)L_P&P Y JOG+
OUT       D002020.5	// L_P&P Y JOG+

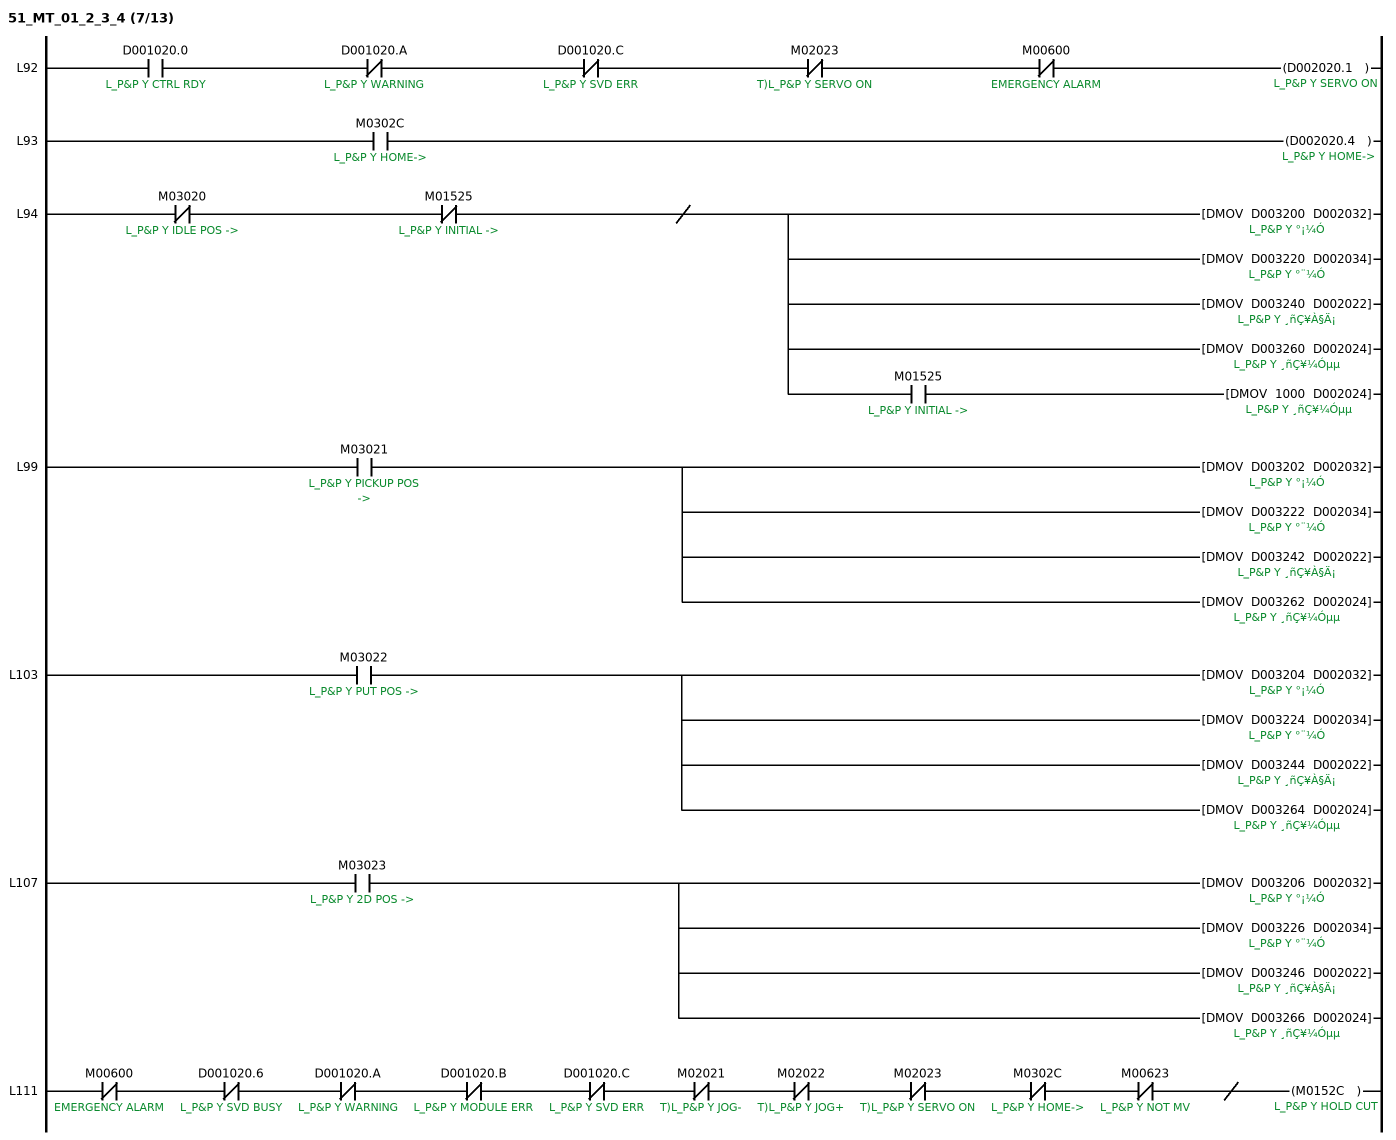
; L92
LOAD      D001020.0	// L_P&P Y CTRL RDY
AND NOT   D001020.A	// L_P&P Y WARNING
AND NOT   D001020.C	// L_P&P Y SVD ERR
AND NOT   M02023	// T)L_P&P Y SERVO ON
AND NOT   M00600	// EMERGENCY ALARM
OUT       D002020.1	// L_P&P Y SERVO ON
; L93
LOAD      M0302C	// L_P&P Y HOME->
OUT       D002020.4	// L_P&P Y HOME->
; L94
LOAD NOT  M03020	// L_P&P Y IDLE POS ->
AND NOT   M01525	// L_P&P Y INITIAL ->
NOT
DMOV      D003200 D002032	// L_P&P Y °¡¼Ó
DMOV      D003220 D002034	// L_P&P Y °¨¼Ó
DMOV      D003240 D002022	// L_P&P Y ¸ñÇ¥À§Ä¡
DMOV      D003260 D002024	// L_P&P Y ¸ñÇ¥¼Óµµ
AND       M01525	// L_P&P Y INITIAL ->
DMOV      1000 D002024	// L_P&P Y ¸ñÇ¥¼Óµµ
; L99
LOAD      M03021	// L_P&P Y PICKUP POS ->
DMOV      D003202 D002032	// L_P&P Y °¡¼Ó
DMOV      D003222 D002034	// L_P&P Y °¨¼Ó
DMOV      D003242 D002022	// L_P&P Y ¸ñÇ¥À§Ä¡
DMOV      D003262 D002024	// L_P&P Y ¸ñÇ¥¼Óµµ
; L103
LOAD      M03022	// L_P&P Y PUT POS ->
DMOV      D003204 D002032	// L_P&P Y °¡¼Ó
DMOV      D003224 D002034	// L_P&P Y °¨¼Ó
DMOV      D003244 D002022	// L_P&P Y ¸ñÇ¥À§Ä¡
DMOV      D003264 D002024	// L_P&P Y ¸ñÇ¥¼Óµµ
; L107
LOAD      M03023	// L_P&P Y 2D POS ->
DMOV      D003206 D002032	// L_P&P Y °¡¼Ó
DMOV      D003226 D002034	// L_P&P Y °¨¼Ó
DMOV      D003246 D002022	// L_P&P Y ¸ñÇ¥À§Ä¡
DMOV      D003266 D002024	// L_P&P Y ¸ñÇ¥¼Óµµ
; L111
LOAD NOT  M00600	// EMERGENCY ALARM
AND NOT   D001020.6	// L_P&P Y SVD BUSY
AND NOT   D001020.A	// L_P&P Y WARNING
AND NOT   D001020.B	// L_P&P Y MODULE ERR
AND NOT   D001020.C	// L_P&P Y SVD ERR
AND NOT   M02021	// T)L_P&P Y JOG-
AND NOT   M02022	// T)L_P&P Y JOG+
AND NOT   M02023	// T)L_P&P Y SERVO ON
AND NOT   M0302C	// L_P&P Y HOME->
AND NOT   M00623	// L_P&P Y NOT MV
NOT
OUT       M0152C	// L_P&P Y HOLD CUT

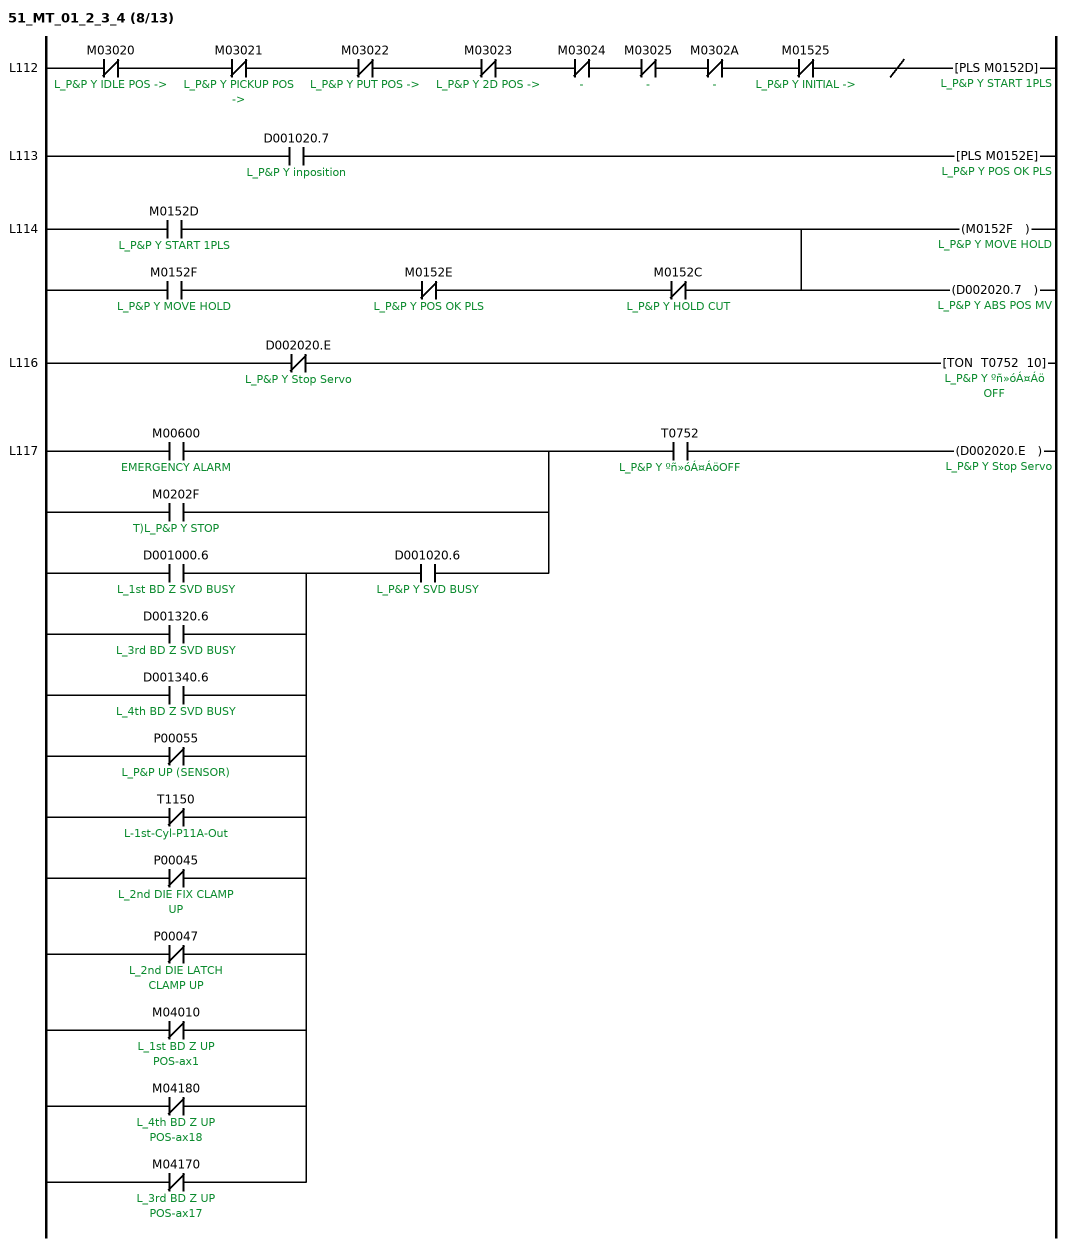
; L112
LOAD NOT  M03020	// L_P&P Y IDLE POS ->
AND NOT   M03021	// L_P&P Y PICKUP POS ->
AND NOT   M03022	// L_P&P Y PUT POS ->
AND NOT   M03023	// L_P&P Y 2D POS ->
AND NOT   M03024	// -
AND NOT   M03025	// -
AND NOT   M0302A	// -
AND NOT   M01525	// L_P&P Y INITIAL ->
NOT
OUTP      M0152D	// L_P&P Y START 1PLS
; L113
LOAD      D001020.7	// L_P&P Y inposition
OUTP      M0152E	// L_P&P Y POS OK PLS
; L114
LOAD      M0152D	// L_P&P Y START 1PLS
LOAD      M0152F	// L_P&P Y MOVE HOLD
AND NOT   M0152E	// L_P&P Y POS OK PLS
AND NOT   M0152C	// L_P&P Y HOLD CUT
OR LOAD
OUT       M0152F	// L_P&P Y MOVE HOLD
OUT       D002020.7	// L_P&P Y ABS POS MV
; L116
LOAD NOT  D002020.E	// L_P&P Y Stop Servo
TON       T0752 10	// L_P&P Y ºñ»óÁ¤ÁöOFF
; L117
LOAD      M00600	// EMERGENCY ALARM
OR        M0202F	// T)L_P&P Y STOP
LOAD      D001000.6	// L_1st BD Z SVD BUSY
OR        D001320.6	// L_3rd BD Z SVD BUSY
OR        D001340.6	// L_4th BD Z SVD BUSY
OR NOT    P00055	// L_P&P UP (SENSOR)
OR NOT    T1150	// L-1st-Cyl-P11A-Out
OR NOT    P00045	// L_2nd DIE FIX CLAMP UP
OR NOT    P00047	// L_2nd DIE LATCH CLAMP UP
OR NOT    M04010	// L_1st BD Z UP POS-ax1
OR NOT    M04180	// L_4th BD Z UP POS-ax18
OR NOT    M04170	// L_3rd BD Z UP POS-ax17
AND       D001020.6	// L_P&P Y SVD BUSY
OR LOAD
AND       T0752	// L_P&P Y ºñ»óÁ¤ÁöOFF
OUT       D002020.E	// L_P&P Y Stop Servo

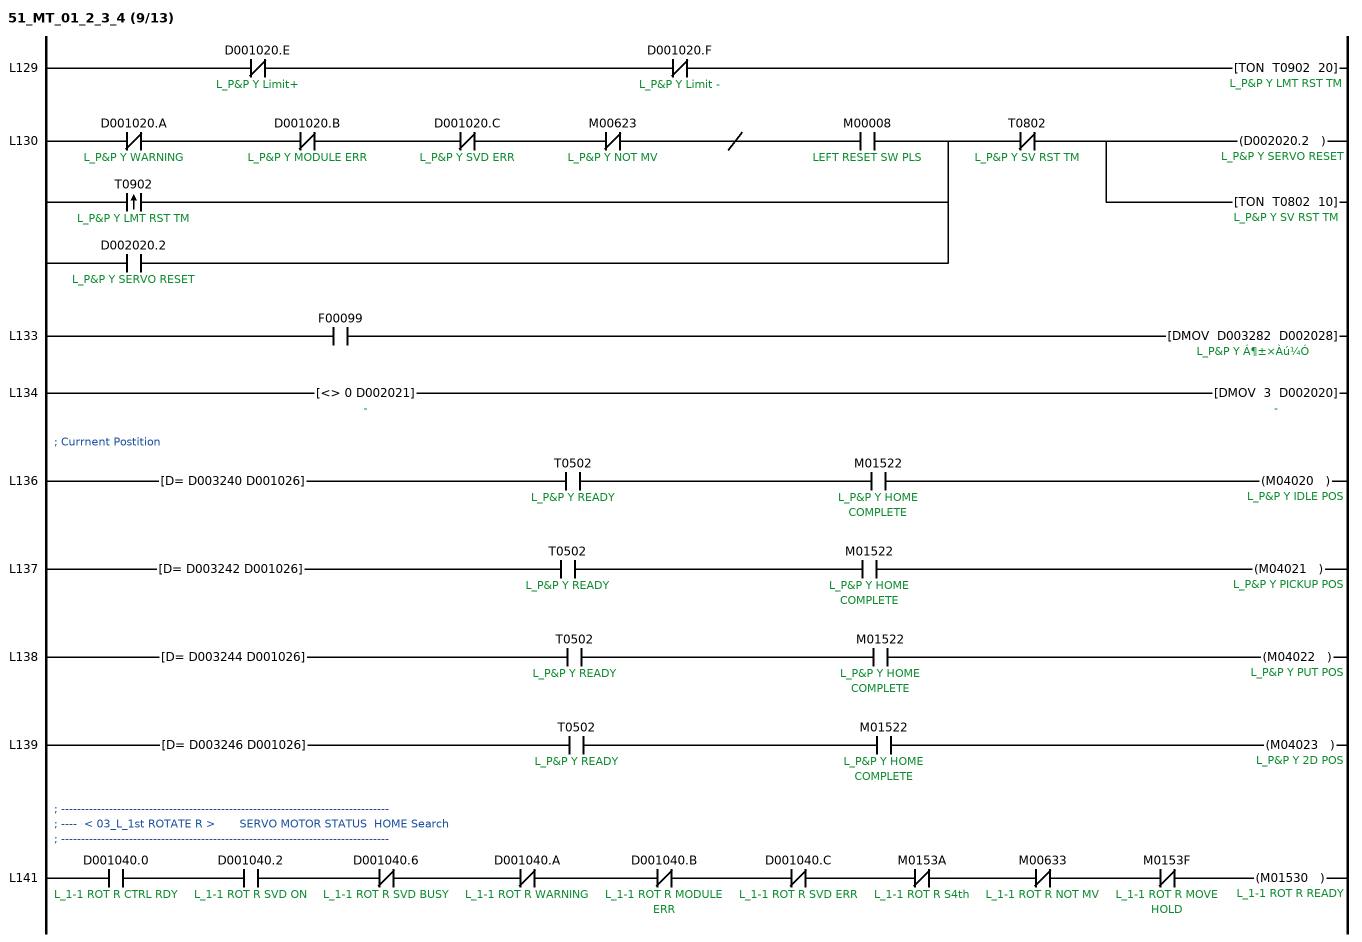
; L129
LOAD NOT  D001020.E	// L_P&P Y Limit+
AND NOT   D001020.F	// L_P&P Y Limit -
TON       T0902 20	// L_P&P Y LMT RST TM
; L130
LOAD NOT  D001020.A	// L_P&P Y WARNING
AND NOT   D001020.B	// L_P&P Y MODULE ERR
AND NOT   D001020.C	// L_P&P Y SVD ERR
AND NOT   M00623	// L_P&P Y NOT MV
NOT
AND       M00008	// LEFT RESET SW PLS
ORP       T0902	// L_P&P Y LMT RST TM
OR        D002020.2	// L_P&P Y SERVO RESET
AND NOT   T0802	// L_P&P Y SV RST TM
OUT       D002020.2	// L_P&P Y SERVO RESET
TON       T0802 10	// L_P&P Y SV RST TM
; L133
LOAD      F00099
DMOV      D003282 D002028	// L_P&P Y Á¶±×Àú¼Ó
; L134
LOAD<>    0 D002021	// -
DMOV      3 D002020	// -
// Currnent Postition
; L136
LOADD=    D003240 D001026
AND       T0502	// L_P&P Y READY
AND       M01522	// L_P&P Y HOME COMPLETE
OUT       M04020	// L_P&P Y IDLE POS
; L137
LOADD=    D003242 D001026
AND       T0502	// L_P&P Y READY
AND       M01522	// L_P&P Y HOME COMPLETE
OUT       M04021	// L_P&P Y PICKUP POS
; L138
LOADD=    D003244 D001026
AND       T0502	// L_P&P Y READY
AND       M01522	// L_P&P Y HOME COMPLETE
OUT       M04022	// L_P&P Y PUT POS
; L139
LOADD=    D003246 D001026
AND       T0502	// L_P&P Y READY
AND       M01522	// L_P&P Y HOME COMPLETE
OUT       M04023	// L_P&P Y 2D POS
// ----------------------------------------------------------------------------------
// 
// ----  < 03_L_1st ROTATE R >       SERVO MOTOR STATUS  HOME Search
// 
// ----------------------------------------------------------------------------------
; L141
LOAD      D001040.0	// L_1-1 ROT R CTRL RDY
AND       D001040.2	// L_1-1 ROT R SVD ON
AND NOT   D001040.6	// L_1-1 ROT R SVD BUSY
AND NOT   D001040.A	// L_1-1 ROT R WARNING
AND NOT   D001040.B	// L_1-1 ROT R MODULE ERR
AND NOT   D001040.C	// L_1-1 ROT R SVD ERR
AND NOT   M0153A	// L_1-1 ROT R S4th
AND NOT   M00633	// L_1-1 ROT R NOT MV
AND NOT   M0153F	// L_1-1 ROT R MOVE HOLD
OUT       M01530	// L_1-1 ROT R READY

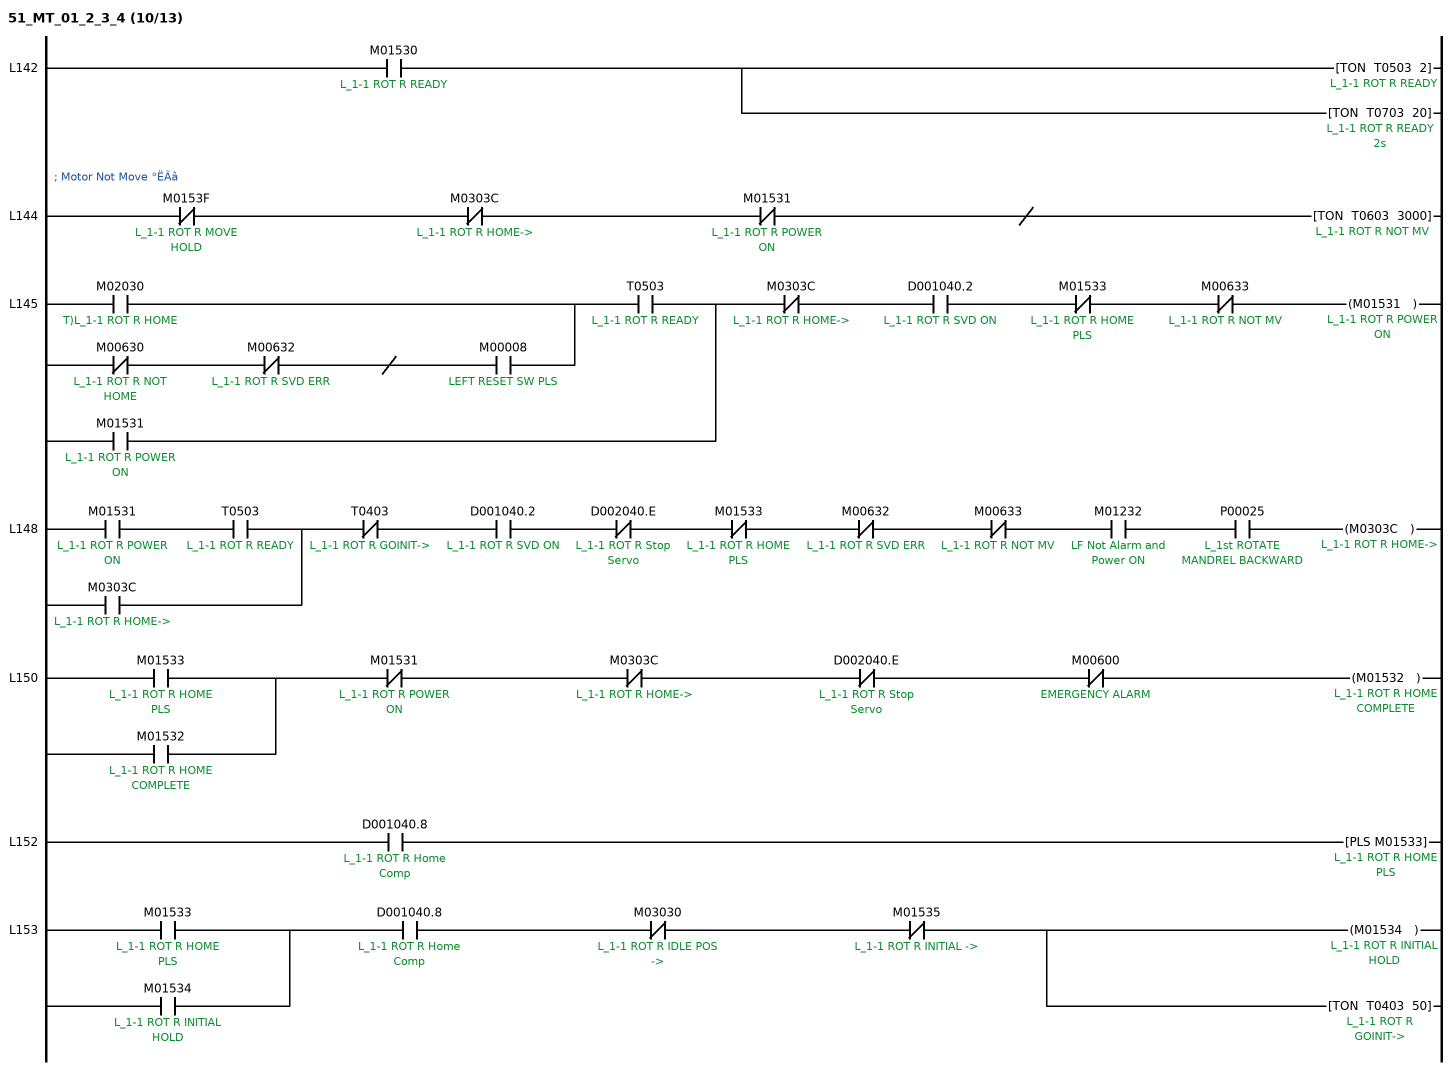
; L142
LOAD      M01530	// L_1-1 ROT R READY
TON       T0503 2	// L_1-1 ROT R READY
TON       T0703 20	// L_1-1 ROT R READY 2s
; L144
LOAD NOT  M0153F	// L_1-1 ROT R MOVE HOLD
AND NOT   M0303C	// L_1-1 ROT R HOME->
AND NOT   M01531	// L_1-1 ROT R POWER ON
NOT
TON       T0603 3000	// L_1-1 ROT R NOT MV
// output comment: Motor Not Move °ËÃâ
; L145
LOAD      M02030	// T)L_1-1 ROT R HOME
LOAD NOT  M00630	// L_1-1 ROT R NOT HOME
AND NOT   M00632	// L_1-1 ROT R SVD ERR
NOT
AND       M00008	// LEFT RESET SW PLS
OR LOAD
AND       T0503	// L_1-1 ROT R READY
OR        M01531	// L_1-1 ROT R POWER ON
AND NOT   M0303C	// L_1-1 ROT R HOME->
AND       D001040.2	// L_1-1 ROT R SVD ON
AND NOT   M01533	// L_1-1 ROT R HOME PLS
AND NOT   M00633	// L_1-1 ROT R NOT MV
OUT       M01531	// L_1-1 ROT R POWER ON
; L148
LOAD      M01531	// L_1-1 ROT R POWER ON
AND       T0503	// L_1-1 ROT R READY
OR        M0303C	// L_1-1 ROT R HOME->
AND NOT   T0403	// L_1-1 ROT R GOINIT->
AND       D001040.2	// L_1-1 ROT R SVD ON
AND NOT   D002040.E	// L_1-1 ROT R Stop Servo
AND NOT   M01533	// L_1-1 ROT R HOME PLS
AND NOT   M00632	// L_1-1 ROT R SVD ERR
AND NOT   M00633	// L_1-1 ROT R NOT MV
AND       M01232	// LF Not Alarm and Power ON
AND       P00025	// L_1st ROTATE MANDREL BACKWARD
OUT       M0303C	// L_1-1 ROT R HOME->
; L150
LOAD      M01533	// L_1-1 ROT R HOME PLS
OR        M01532	// L_1-1 ROT R HOME COMPLETE
AND NOT   M01531	// L_1-1 ROT R POWER ON
AND NOT   M0303C	// L_1-1 ROT R HOME->
AND NOT   D002040.E	// L_1-1 ROT R Stop Servo
AND NOT   M00600	// EMERGENCY ALARM
OUT       M01532	// L_1-1 ROT R HOME COMPLETE
; L152
LOAD      D001040.8	// L_1-1 ROT R Home Comp 
OUTP      M01533	// L_1-1 ROT R HOME PLS
; L153
LOAD      M01533	// L_1-1 ROT R HOME PLS
OR        M01534	// L_1-1 ROT R INITIAL HOLD
AND       D001040.8	// L_1-1 ROT R Home Comp 
AND NOT   M03030	// L_1-1 ROT R IDLE POS ->
AND NOT   M01535	// L_1-1 ROT R INITIAL ->
OUT       M01534	// L_1-1 ROT R INITIAL HOLD
TON       T0403 50	// L_1-1 ROT R GOINIT->

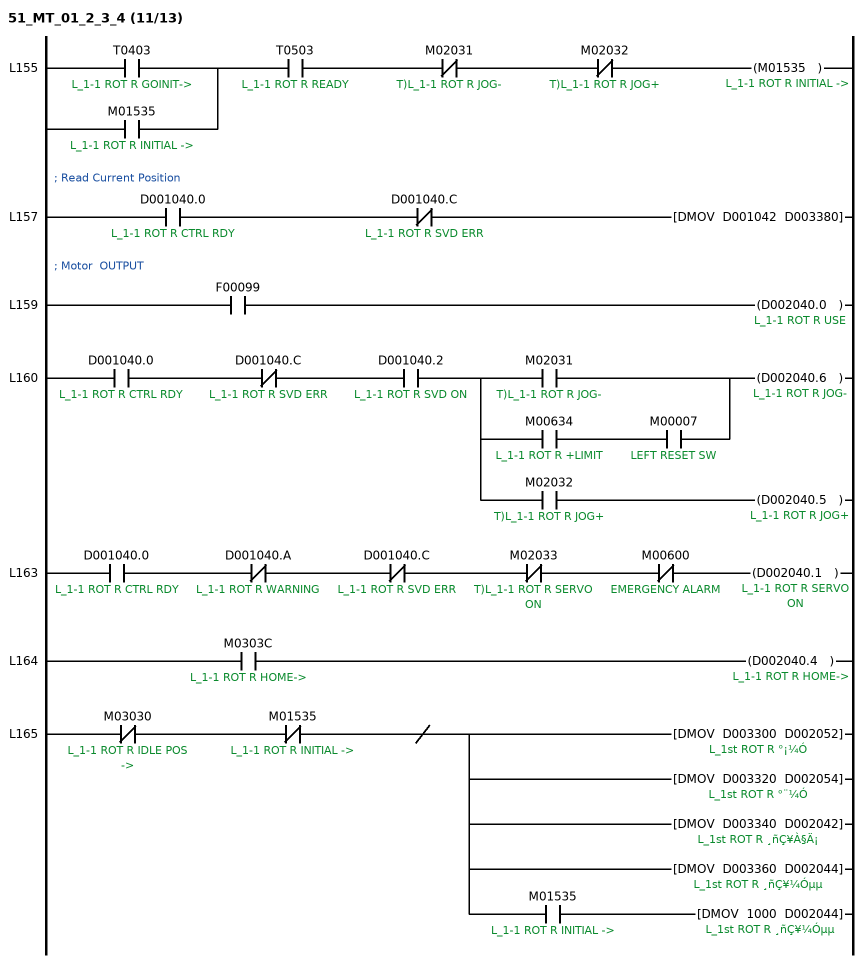
; L155
LOAD      T0403	// L_1-1 ROT R GOINIT->
OR        M01535	// L_1-1 ROT R INITIAL ->
AND       T0503	// L_1-1 ROT R READY
AND NOT   M02031	// T)L_1-1 ROT R JOG-
AND NOT   M02032	// T)L_1-1 ROT R JOG+
OUT       M01535	// L_1-1 ROT R INITIAL ->
; L157
LOAD      D001040.0	// L_1-1 ROT R CTRL RDY
AND NOT   D001040.C	// L_1-1 ROT R SVD ERR
DMOV      D001042 D003380
// output comment: Read Current Position
//  Motor  OUTPUT
; L159
LOAD      F00099
OUT       D002040.0	// L_1-1 ROT R USE
; L160
LOAD      D001040.0	// L_1-1 ROT R CTRL RDY
AND NOT   D001040.C	// L_1-1 ROT R SVD ERR
AND       D001040.2	// L_1-1 ROT R SVD ON
MPUSH
LOAD      M02031	// T)L_1-1 ROT R JOG-
LOAD      M00634	// L_1-1 ROT R +LIMIT
AND       M00007	// LEFT RESET SW
OR LOAD
AND LOAD
OUT       D002040.6	// L_1-1 ROT R JOG-
MPOP
AND       M02032	// T)L_1-1 ROT R JOG+
OUT       D002040.5	// L_1-1 ROT R JOG+
; L163
LOAD      D001040.0	// L_1-1 ROT R CTRL RDY
AND NOT   D001040.A	// L_1-1 ROT R WARNING
AND NOT   D001040.C	// L_1-1 ROT R SVD ERR
AND NOT   M02033	// T)L_1-1 ROT R SERVO ON
AND NOT   M00600	// EMERGENCY ALARM
OUT       D002040.1	// L_1-1 ROT R SERVO ON
; L164
LOAD      M0303C	// L_1-1 ROT R HOME->
OUT       D002040.4	// L_1-1 ROT R HOME->
; L165
LOAD NOT  M03030	// L_1-1 ROT R IDLE POS ->
AND NOT   M01535	// L_1-1 ROT R INITIAL ->
NOT
DMOV      D003300 D002052	// L_1st ROT R °¡¼Ó
DMOV      D003320 D002054	// L_1st ROT R °¨¼Ó
DMOV      D003340 D002042	// L_1st ROT R ¸ñÇ¥À§Ä¡
DMOV      D003360 D002044	// L_1st ROT R ¸ñÇ¥¼Óµµ
AND       M01535	// L_1-1 ROT R INITIAL ->
DMOV      1000 D002044	// L_1st ROT R ¸ñÇ¥¼Óµµ

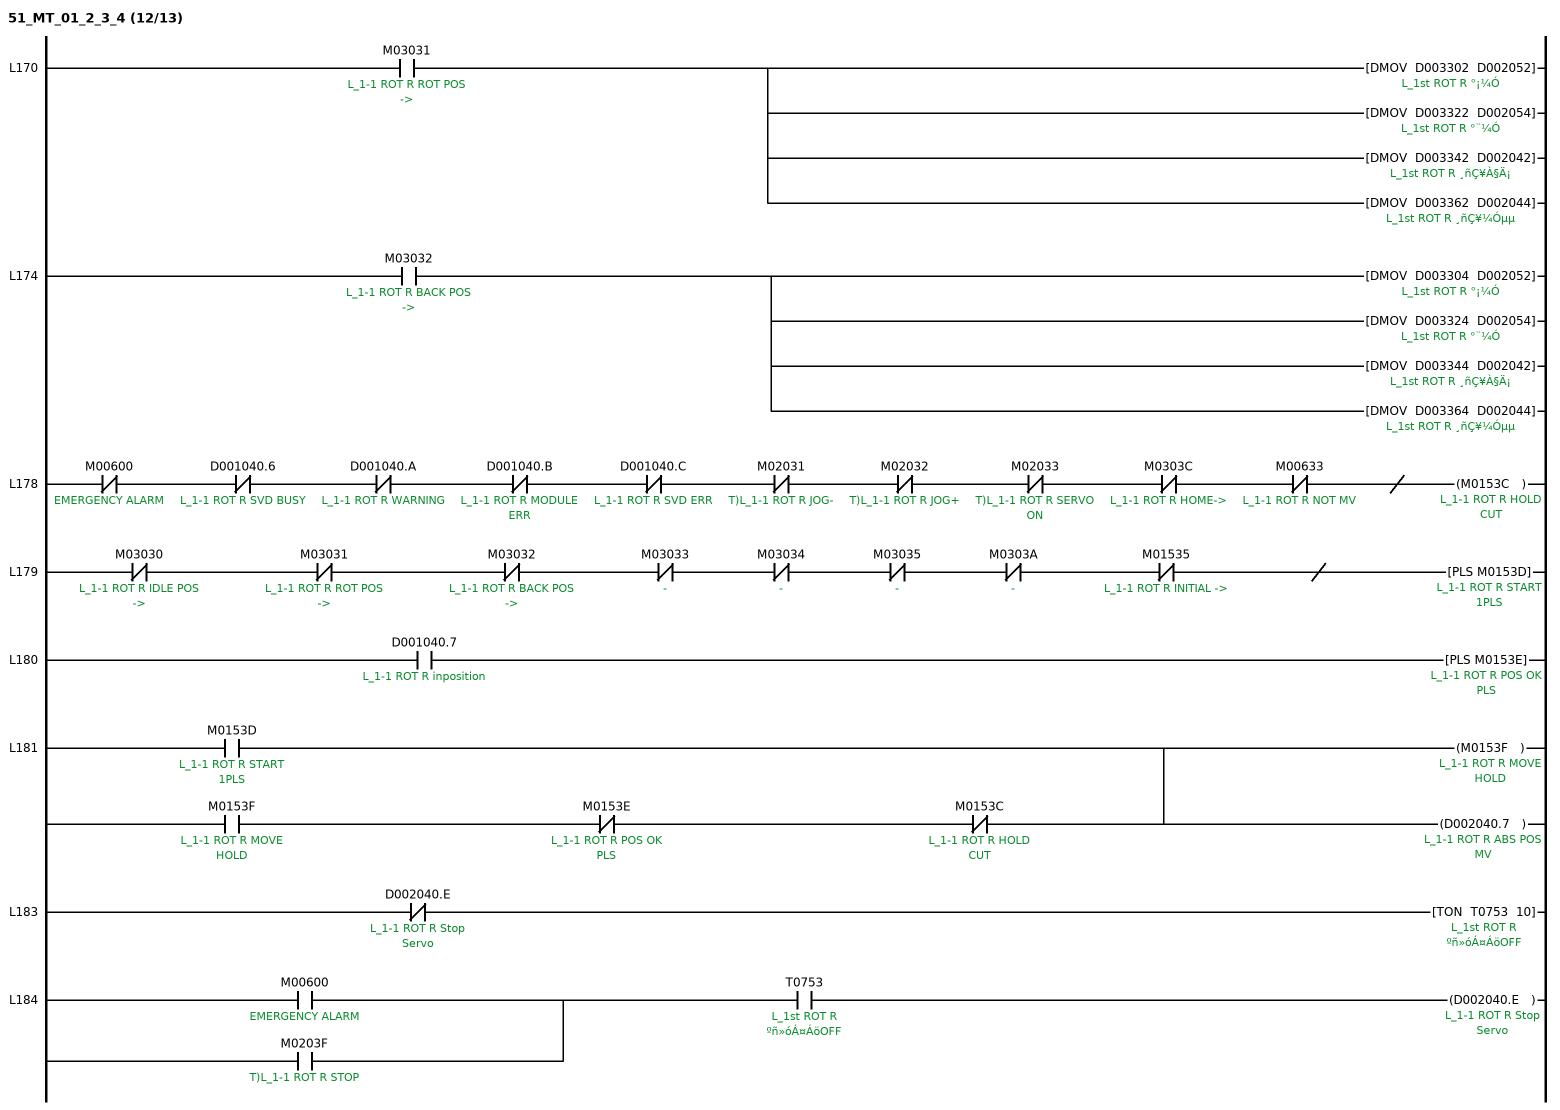
; L170
LOAD      M03031	// L_1-1 ROT R ROT POS ->
DMOV      D003302 D002052	// L_1st ROT R °¡¼Ó
DMOV      D003322 D002054	// L_1st ROT R °¨¼Ó
DMOV      D003342 D002042	// L_1st ROT R ¸ñÇ¥À§Ä¡
DMOV      D003362 D002044	// L_1st ROT R ¸ñÇ¥¼Óµµ
; L174
LOAD      M03032	// L_1-1 ROT R BACK POS ->
DMOV      D003304 D002052	// L_1st ROT R °¡¼Ó
DMOV      D003324 D002054	// L_1st ROT R °¨¼Ó
DMOV      D003344 D002042	// L_1st ROT R ¸ñÇ¥À§Ä¡
DMOV      D003364 D002044	// L_1st ROT R ¸ñÇ¥¼Óµµ
; L178
LOAD NOT  M00600	// EMERGENCY ALARM
AND NOT   D001040.6	// L_1-1 ROT R SVD BUSY
AND NOT   D001040.A	// L_1-1 ROT R WARNING
AND NOT   D001040.B	// L_1-1 ROT R MODULE ERR
AND NOT   D001040.C	// L_1-1 ROT R SVD ERR
AND NOT   M02031	// T)L_1-1 ROT R JOG-
AND NOT   M02032	// T)L_1-1 ROT R JOG+
AND NOT   M02033	// T)L_1-1 ROT R SERVO ON
AND NOT   M0303C	// L_1-1 ROT R HOME->
AND NOT   M00633	// L_1-1 ROT R NOT MV
NOT
OUT       M0153C	// L_1-1 ROT R HOLD CUT
; L179
LOAD NOT  M03030	// L_1-1 ROT R IDLE POS ->
AND NOT   M03031	// L_1-1 ROT R ROT POS ->
AND NOT   M03032	// L_1-1 ROT R BACK POS ->
AND NOT   M03033	// -
AND NOT   M03034	// -
AND NOT   M03035	// -
AND NOT   M0303A	// -
AND NOT   M01535	// L_1-1 ROT R INITIAL ->
NOT
OUTP      M0153D	// L_1-1 ROT R START 1PLS
; L180
LOAD      D001040.7	// L_1-1 ROT R inposition
OUTP      M0153E	// L_1-1 ROT R POS OK PLS
; L181
LOAD      M0153D	// L_1-1 ROT R START 1PLS
LOAD      M0153F	// L_1-1 ROT R MOVE HOLD
AND NOT   M0153E	// L_1-1 ROT R POS OK PLS
AND NOT   M0153C	// L_1-1 ROT R HOLD CUT
OR LOAD
OUT       M0153F	// L_1-1 ROT R MOVE HOLD
OUT       D002040.7	// L_1-1 ROT R ABS POS MV
; L183
LOAD NOT  D002040.E	// L_1-1 ROT R Stop Servo
TON       T0753 10	// L_1st ROT R ºñ»óÁ¤ÁöOFF
; L184
LOAD      M00600	// EMERGENCY ALARM
OR        M0203F	// T)L_1-1 ROT R STOP
AND       T0753	// L_1st ROT R ºñ»óÁ¤ÁöOFF
OUT       D002040.E	// L_1-1 ROT R Stop Servo

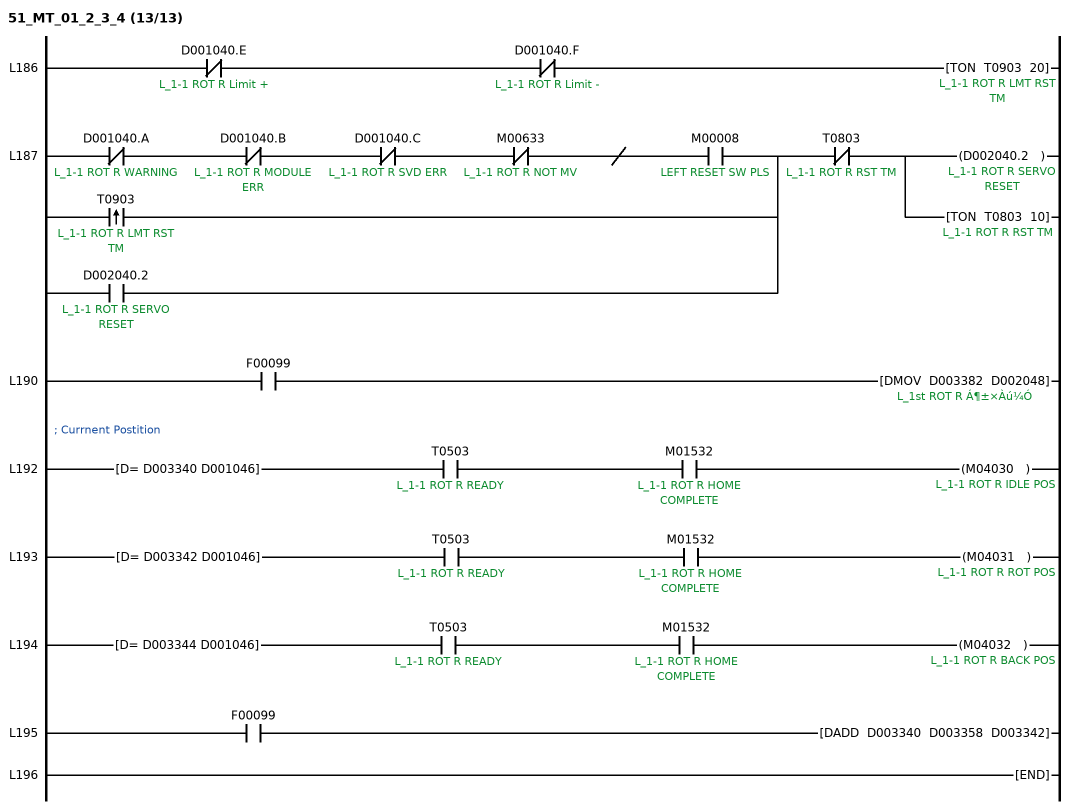
; L186
LOAD NOT  D001040.E	// L_1-1 ROT R Limit +
AND NOT   D001040.F	// L_1-1 ROT R Limit -
TON       T0903 20	// L_1-1 ROT R LMT RST TM
; L187
LOAD NOT  D001040.A	// L_1-1 ROT R WARNING
AND NOT   D001040.B	// L_1-1 ROT R MODULE ERR
AND NOT   D001040.C	// L_1-1 ROT R SVD ERR
AND NOT   M00633	// L_1-1 ROT R NOT MV
NOT
AND       M00008	// LEFT RESET SW PLS
ORP       T0903	// L_1-1 ROT R LMT RST TM
OR        D002040.2	// L_1-1 ROT R SERVO RESET
AND NOT   T0803	// L_1-1 ROT R RST TM
OUT       D002040.2	// L_1-1 ROT R SERVO RESET
TON       T0803 10	// L_1-1 ROT R RST TM
; L190
LOAD      F00099
DMOV      D003382 D002048	// L_1st ROT R Á¶±×Àú¼Ó
// Currnent Postition
; L192
LOADD=    D003340 D001046
AND       T0503	// L_1-1 ROT R READY
AND       M01532	// L_1-1 ROT R HOME COMPLETE
OUT       M04030	// L_1-1 ROT R IDLE POS
; L193
LOADD=    D003342 D001046
AND       T0503	// L_1-1 ROT R READY
AND       M01532	// L_1-1 ROT R HOME COMPLETE
OUT       M04031	// L_1-1 ROT R ROT POS
; L194
LOADD=    D003344 D001046
AND       T0503	// L_1-1 ROT R READY
AND       M01532	// L_1-1 ROT R HOME COMPLETE
OUT       M04032	// L_1-1 ROT R BACK POS
; L195
LOAD      F00099
DADD      D003340 D003358 D003342
; L196
END

PROGRAM 52_MT_05_6_7_8 (task: ½ºÄµ ÇÁ·Î±×·¥)

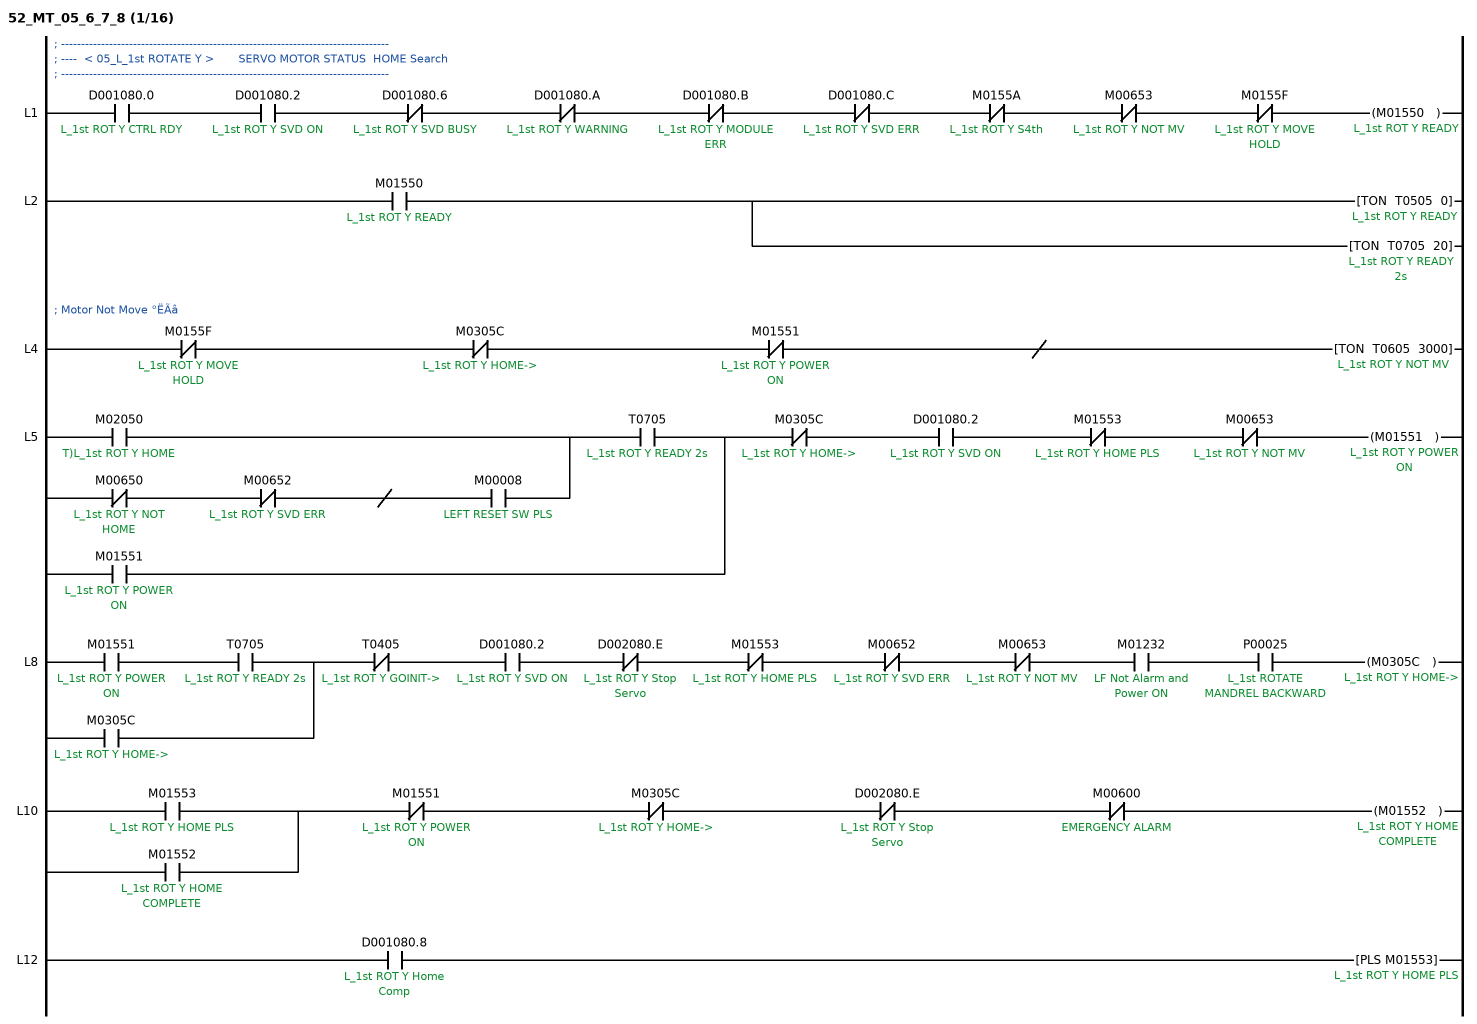
// ----------------------------------------------------------------------------------
// 
// ----  < 05_L_1st ROTATE Y >       SERVO MOTOR STATUS  HOME Search
// 
// ----------------------------------------------------------------------------------
; L1
LOAD      D001080.0	// L_1st ROT Y CTRL RDY
AND       D001080.2	// L_1st ROT Y SVD ON
AND NOT   D001080.6	// L_1st ROT Y SVD BUSY
AND NOT   D001080.A	// L_1st ROT Y WARNING
AND NOT   D001080.B	// L_1st ROT Y MODULE ERR
AND NOT   D001080.C	// L_1st ROT Y SVD ERR
AND NOT   M0155A	// L_1st ROT Y S4th
AND NOT   M00653	// L_1st ROT Y NOT MV
AND NOT   M0155F	// L_1st ROT Y MOVE HOLD
OUT       M01550	// L_1st ROT Y READY
; L2
LOAD      M01550	// L_1st ROT Y READY
TON       T0505 0	// L_1st ROT Y READY
TON       T0705 20	// L_1st ROT Y READY 2s
; L4
LOAD NOT  M0155F	// L_1st ROT Y MOVE HOLD
AND NOT   M0305C	// L_1st ROT Y HOME->
AND NOT   M01551	// L_1st ROT Y POWER ON
NOT
TON       T0605 3000	// L_1st ROT Y NOT MV
// output comment: Motor Not Move °ËÃâ
; L5
LOAD      M02050	// T)L_1st ROT Y HOME
LOAD NOT  M00650	// L_1st ROT Y NOT HOME
AND NOT   M00652	// L_1st ROT Y SVD ERR
NOT
AND       M00008	// LEFT RESET SW PLS
OR LOAD
AND       T0705	// L_1st ROT Y READY 2s
OR        M01551	// L_1st ROT Y POWER ON
AND NOT   M0305C	// L_1st ROT Y HOME->
AND       D001080.2	// L_1st ROT Y SVD ON
AND NOT   M01553	// L_1st ROT Y HOME PLS
AND NOT   M00653	// L_1st ROT Y NOT MV
OUT       M01551	// L_1st ROT Y POWER ON
; L8
LOAD      M01551	// L_1st ROT Y POWER ON
AND       T0705	// L_1st ROT Y READY 2s
OR        M0305C	// L_1st ROT Y HOME->
AND NOT   T0405	// L_1st ROT Y GOINIT->
AND       D001080.2	// L_1st ROT Y SVD ON
AND NOT   D002080.E	// L_1st ROT Y Stop Servo
AND NOT   M01553	// L_1st ROT Y HOME PLS
AND NOT   M00652	// L_1st ROT Y SVD ERR
AND NOT   M00653	// L_1st ROT Y NOT MV
AND       M01232	// LF Not Alarm and Power ON
AND       P00025	// L_1st ROTATE MANDREL BACKWARD
OUT       M0305C	// L_1st ROT Y HOME->
; L10
LOAD      M01553	// L_1st ROT Y HOME PLS
OR        M01552	// L_1st ROT Y HOME COMPLETE
AND NOT   M01551	// L_1st ROT Y POWER ON
AND NOT   M0305C	// L_1st ROT Y HOME->
AND NOT   D002080.E	// L_1st ROT Y Stop Servo
AND NOT   M00600	// EMERGENCY ALARM
OUT       M01552	// L_1st ROT Y HOME COMPLETE
; L12
LOAD      D001080.8	// L_1st ROT Y Home Comp
OUTP      M01553	// L_1st ROT Y HOME PLS

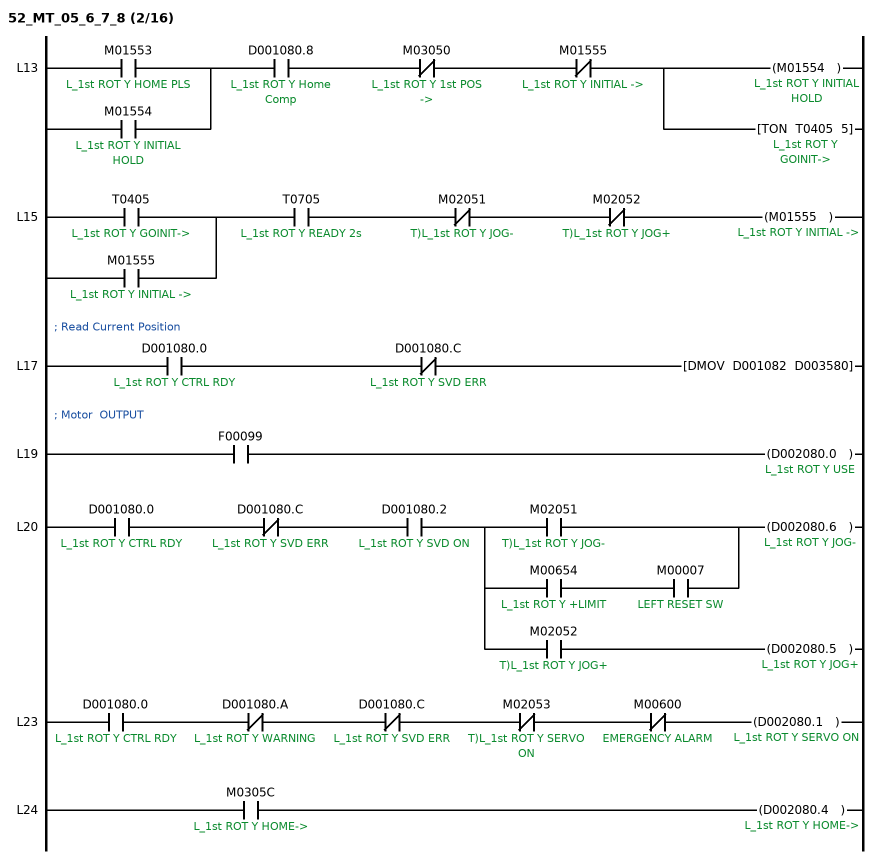
; L13
LOAD      M01553	// L_1st ROT Y HOME PLS
OR        M01554	// L_1st ROT Y INITIAL HOLD
AND       D001080.8	// L_1st ROT Y Home Comp
AND NOT   M03050	// L_1st ROT Y 1st POS ->
AND NOT   M01555	// L_1st ROT Y INITIAL ->
OUT       M01554	// L_1st ROT Y INITIAL HOLD
TON       T0405 5	// L_1st ROT Y GOINIT->
; L15
LOAD      T0405	// L_1st ROT Y GOINIT->
OR        M01555	// L_1st ROT Y INITIAL ->
AND       T0705	// L_1st ROT Y READY 2s
AND NOT   M02051	// T)L_1st ROT Y JOG-
AND NOT   M02052	// T)L_1st ROT Y JOG+
OUT       M01555	// L_1st ROT Y INITIAL ->
; L17
LOAD      D001080.0	// L_1st ROT Y CTRL RDY
AND NOT   D001080.C	// L_1st ROT Y SVD ERR
DMOV      D001082 D003580
// output comment: Read Current Position
//  Motor  OUTPUT
; L19
LOAD      F00099
OUT       D002080.0	// L_1st ROT Y USE
; L20
LOAD      D001080.0	// L_1st ROT Y CTRL RDY
AND NOT   D001080.C	// L_1st ROT Y SVD ERR
AND       D001080.2	// L_1st ROT Y SVD ON
MPUSH
LOAD      M02051	// T)L_1st ROT Y JOG-
LOAD      M00654	// L_1st ROT Y +LIMIT
AND       M00007	// LEFT RESET SW
OR LOAD
AND LOAD
OUT       D002080.6	// L_1st ROT Y JOG-
MPOP
AND       M02052	// T)L_1st ROT Y JOG+
OUT       D002080.5	// L_1st ROT Y JOG+
; L23
LOAD      D001080.0	// L_1st ROT Y CTRL RDY
AND NOT   D001080.A	// L_1st ROT Y WARNING
AND NOT   D001080.C	// L_1st ROT Y SVD ERR
AND NOT   M02053	// T)L_1st ROT Y SERVO ON
AND NOT   M00600	// EMERGENCY ALARM
OUT       D002080.1	// L_1st ROT Y SERVO ON
; L24
LOAD      M0305C	// L_1st ROT Y HOME->
OUT       D002080.4	// L_1st ROT Y HOME->

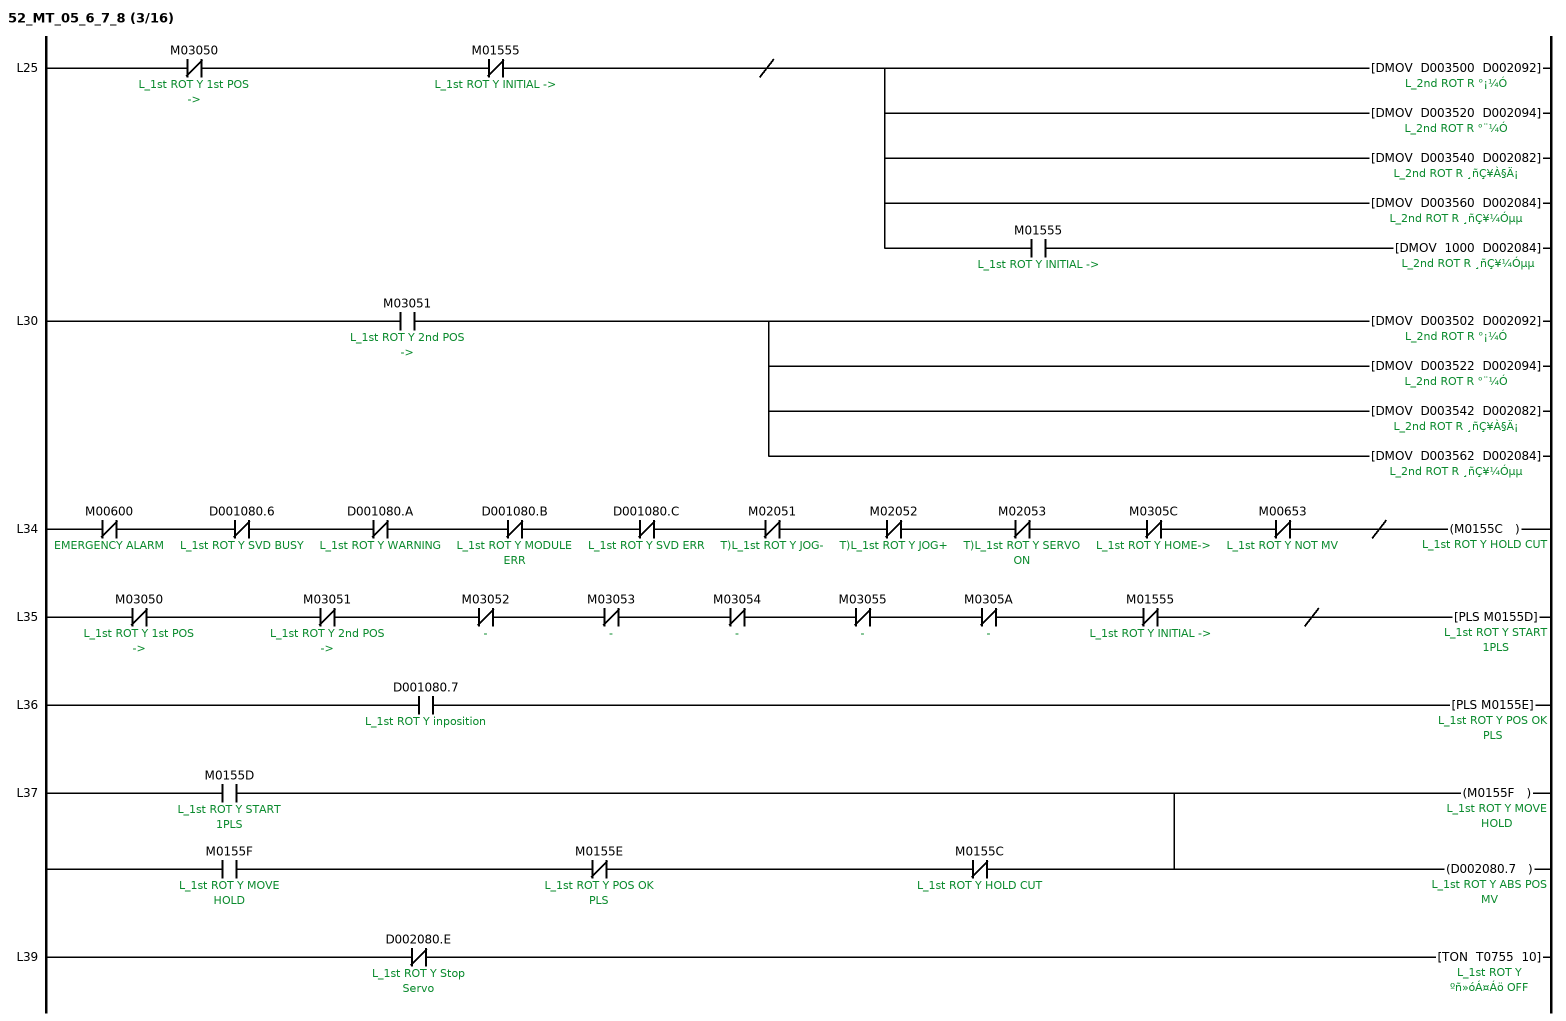
; L25
LOAD NOT  M03050	// L_1st ROT Y 1st POS ->
AND NOT   M01555	// L_1st ROT Y INITIAL ->
NOT
DMOV      D003500 D002092	// L_2nd ROT R °¡¼Ó
DMOV      D003520 D002094	// L_2nd ROT R °¨¼Ó
DMOV      D003540 D002082	// L_2nd ROT R ¸ñÇ¥À§Ä¡
DMOV      D003560 D002084	// L_2nd ROT R ¸ñÇ¥¼Óµµ
AND       M01555	// L_1st ROT Y INITIAL ->
DMOV      1000 D002084	// L_2nd ROT R ¸ñÇ¥¼Óµµ
; L30
LOAD      M03051	// L_1st ROT Y 2nd POS ->
DMOV      D003502 D002092	// L_2nd ROT R °¡¼Ó
DMOV      D003522 D002094	// L_2nd ROT R °¨¼Ó
DMOV      D003542 D002082	// L_2nd ROT R ¸ñÇ¥À§Ä¡
DMOV      D003562 D002084	// L_2nd ROT R ¸ñÇ¥¼Óµµ
; L34
LOAD NOT  M00600	// EMERGENCY ALARM
AND NOT   D001080.6	// L_1st ROT Y SVD BUSY
AND NOT   D001080.A	// L_1st ROT Y WARNING
AND NOT   D001080.B	// L_1st ROT Y MODULE ERR
AND NOT   D001080.C	// L_1st ROT Y SVD ERR
AND NOT   M02051	// T)L_1st ROT Y JOG-
AND NOT   M02052	// T)L_1st ROT Y JOG+
AND NOT   M02053	// T)L_1st ROT Y SERVO ON
AND NOT   M0305C	// L_1st ROT Y HOME->
AND NOT   M00653	// L_1st ROT Y NOT MV
NOT
OUT       M0155C	// L_1st ROT Y HOLD CUT
; L35
LOAD NOT  M03050	// L_1st ROT Y 1st POS ->
AND NOT   M03051	// L_1st ROT Y 2nd POS ->
AND NOT   M03052	// -
AND NOT   M03053	// -
AND NOT   M03054	// -
AND NOT   M03055	// -
AND NOT   M0305A	// -
AND NOT   M01555	// L_1st ROT Y INITIAL ->
NOT
OUTP      M0155D	// L_1st ROT Y START 1PLS
; L36
LOAD      D001080.7	// L_1st ROT Y inposition
OUTP      M0155E	// L_1st ROT Y POS OK PLS
; L37
LOAD      M0155D	// L_1st ROT Y START 1PLS
LOAD      M0155F	// L_1st ROT Y MOVE HOLD
AND NOT   M0155E	// L_1st ROT Y POS OK PLS
AND NOT   M0155C	// L_1st ROT Y HOLD CUT
OR LOAD
OUT       M0155F	// L_1st ROT Y MOVE HOLD
OUT       D002080.7	// L_1st ROT Y ABS POS MV
; L39
LOAD NOT  D002080.E	// L_1st ROT Y Stop Servo
TON       T0755 10	// L_1st ROT Y ºñ»óÁ¤Áö OFF

